# B&R Automation Studio project RS15_RX_30005_r00 (part 4)

#### FP_HeaterInit.st
```iecst
(********************************************************************
 * COPYRIGHT -- .
 ********************************************************************
 * Program: FP_Heater
 * File: FP_HeaterInit.st
 * Author: dominique
 * Created: August 22, 2012
 ********************************************************************
 * Implementation of program FP_Heater
 ********************************************************************)

PROGRAM _INIT

  rPT1_t                   := 25 ;
  rDeltaTStopPicChauf      := 68 ;
  rSeuilConsTempActBattTOR := 132.8 ;

  rPIDRegTChaufKP[1] := 18 ;
  rPIDRegTChaufKI[1] := 30 ;
  rPIDRegTChaufKD[1] := 1 ;

END_PROGRAM
```

### Program Logical/BagMachine_Section/GlobProgCalc (IEC)

#### GlobProgCalcCyclic.st - Cyclic code
```iecst
(********************************************************************
 * COPYRIGHT -- .
 ********************************************************************
 * Program: GlobProgCalc
 * File: GlobProgCalcCyclic.st
 * Author: dominique
 * Created: October 27, 2011
 ********************************************************************
 * Implementation of program GlobProgCalc
 ********************************************************************)

PROGRAM _CYCLIC
// --------------------------------------------------------------------------------------------------
  // Tube Length Limit

  CASE g_iMachType OF
    C_iRS15 :
      g_rMaxBagSize_Inch := g_rMaxBagSize_RS15_mm / 25.4 ;
      g_rMinBagSize_Inch := g_rMinBagSize_RS15_mm / 25.4 ;
    C_iRS26 :
      IF gRecipeActive.bSelEnvBProd THEN
        // Case Envelope Bag
        g_rMaxBagSize_Inch := g_rMaxBagSize_EnvB_mm / 25.4 ;
        g_rMinBagSize_Inch := g_rMinBagSize_EnvB_mm / 25.4 ;
      ELSE
        g_rMaxBagSize_Inch := g_rMaxBagSize_RS26_mm / 25.4 ;
        g_rMinBagSize_Inch := g_rMinBagSize_RS26_mm / 25.4 ;
      END_IF ;
  END_CASE ;

  // Limit operator setting in case of Flexo Type
  gRecipeActive.iPrintUp := LIMIT(1,gRecipeActive.iPrintUp,4) ;
  gRecipeActive.Repeat := LIMIT(g_rMinBagSize_Inch,gRecipeActive.Repeat,g_rMaxBagSize_Inch) ;

  // Repeat calculation in case of Flexo Press
  rPrintUp := INT_TO_REAL(gRecipeActive.iPrintUp) ; // Number of pictures per round of printing cylinder
  CASE g_iFlexoType OF
    C_iM : ; // Case Metric
      iNmaxTooth := TRUNC(g_rMaxBagSize_Inch*25.4/10.0) ;
      iNminTooth := TRUNC(g_rMinBagSize_Inch*25.4/10.0) ;
      IF gRecipeActive.bSelFPProd THEN
        gRecipeActive.Repeat := TRUNC(gRecipeActive.iNumToothGearPrint*10.0)/25.4/rPrintUp ;
      ELSE
        // treatment imperfection calculation of number of tooth otherwise 600mm give 59 tooth instead of 60
        rRepeatMetric := gRecipeActive.Repeat * 25.4 ;
        rRepMet_DecPart := rRepeatMetric - TRUNC(rRepeatMetric) ;
        IF rRepMet_DecPart > 0.5 THEN
          gRecipeActive.iNumToothGearPrint := TRUNC(rRepeatMetric/10.0) + 1 ;
        ELSE
          gRecipeActive.iNumToothGearPrint := TRUNC(rRepeatMetric/10.0) ;
        END_IF ;
      END_IF
      gRecipeActive.iNumToothGearPrint := LIMIT(iNminTooth,gRecipeActive.iNumToothGearPrint,iNmaxTooth) ;
    C_i8DP : ; // Case 8DP
      iNmaxTooth := TRUNC(g_rMaxBagSize_Inch/3.14*8.0) ;
      iNminTooth := TRUNC(g_rMinBagSize_Inch/3.14*8.0) ;
      IF gRecipeActive.bSelFPProd THEN
        gRecipeActive.Repeat := TRUNC(gRecipeActive.iNumToothGearPrint*PI/8.0*1000.0)/1000.0/rPrintUp ;
      ELSE
        gRecipeActive.iNumToothGearPrint := TRUNC(gRecipeActive.Repeat/3.14*8.0) ;
      END_IF
      gRecipeActive.iNumToothGearPrint := LIMIT(iNminTooth,gRecipeActive.iNumToothGearPrint,iNmaxTooth) ;
    C_i10DP : ; // Case 10DP
      iNmaxTooth := TRUNC(g_rMaxBagSize_Inch/3.14*10.0) ;
      iNminTooth := TRUNC(g_rMinBagSize_Inch/3.14*10.0) ;
      IF gRecipeActive.bSelFPProd THEN
        gRecipeActive.Repeat := TRUNC(gRecipeActive.iNumToothGearPrint*PI/10.0*1000.0)/1000.0/rPrintUp ;
      ELSE
        gRecipeActive.iNumToothGearPrint := TRUNC(gRecipeActive.Repeat/3.14*10.0) ;
      END_IF
      gRecipeActive.iNumToothGearPrint := LIMIT(iNminTooth,gRecipeActive.iNumToothGearPrint,iNmaxTooth) ;
    C_i1_4P : ; // Case 1/4"
      iNmaxTooth := TRUNC(g_rMaxBagSize_Inch*4.0) ;
      iNminTooth := TRUNC(g_rMinBagSize_Inch*4.0)+1 ; // D.M. 16/11/2011 RS26 BrownPaper_14606 +1 otherwise minimum tube lentgth = 159mm insted of 160mm and it important for the synchro ratio of the Holding Axis lower than tube length 160mm the Holding Axis makes 1/4 round per bag => not correct for RS26
      IF gRecipeActive.bSelFPProd THEN
        gRecipeActive.Repeat := TRUNC(gRecipeActive.iNumToothGearPrint/4.0*1000.0)/1000.0/rPrintUp ;
      ELSE
        gRecipeActive.iNumToothGearPrint := TRUNC(gRecipeActive.Repeat*4.0) ;
      END_IF
      gRecipeActive.iNumToothGearPrint := LIMIT(iNminTooth,gRecipeActive.iNumToothGearPrint,iNmaxTooth) ;
  END_CASE

// --------------------------------------------------------------------------------------------------
  // Synchro axis OK
  g_bSynchroAxisOK := ( gA[1].Ind_bSynchroOK  AND
                        gA[11].Ind_bSynchroOK OR
                        NOT(gPerf_On) )       AND
                      ( gA[2].Ind_bSynchroOK  OR
                        NOT(gA[2].bActive) )  AND
                      gA[3].Ind_bSynchroOK    AND
                      gA[4].Ind_bSynchroOK    AND
                      gA[5].Ind_bSynchroOK    AND
                      gA[6].Ind_bSynchroOK    AND
                      gA[7].Ind_bSynchroOK    AND
                      ( gA[8].Ind_bSynchroOK  OR
                        NOT(gA[8].bActive) )  AND
                      ( gA[12].Ind_bSynchroOK OR
                        NOT(gA[12].bInMach) ) AND
                      ( gA[13].Ind_bSynchroOK OR
                        NOT(gA[13].bInMach) ) AND
                      1                       ;
  // Synchro axis in progress
  g_bSynchroAxisInProgress := gA[9].Ind_InMotion    AND
                              NOT(g_bSynchroAxisOK) ;
  //
  // Synchro Holding, Tearing and Drum axis
  g_bIndSynchroHTD_OK := gA[3].Ind_bSynchroOK    AND
                         gA[4].Ind_bSynchroOK    AND
                         gA[7].Ind_bSynchroOK    AND
                         ( gA[12].Ind_bSynchroOK OR
                           NOT(gA[12].bInMach) ) AND
                         ( gA[13].Ind_bSynchroOK OR
                           NOT(gA[13].bInMach) ) ;

// --------------------------------------------------------------------------------------------------
  g_bCycManTimeSetOn := gstCycA[1].CycManTimSet.bSCyc  OR
                        gstCycA[3].CycManTimSet.bSCyc  OR
                        gstCycA[4].CycManTimSet.bSCyc  OR
                        gstCycA[7].CycManTimSet.bSCyc  OR
                        gstCycA[12].CycManTimSet.bSCyc AND
                        gA[12].bInMach                 OR
                        gstCycA[13].CycManTimSet.bSCyc AND
                        gA[13].bInMach                 OR
                        0                              ;
END_PROGRAM
```

#### GlobProgCalc.var - Local variables
```iecst
(********************************************************************
 * COPYRIGHT -- .
 ********************************************************************
 * Program: GlobProgCalc
 * File: GlobProgCalc.var
 * Author: dominique
 * Created: October 27, 2011
 ********************************************************************
 * Local variables of program GlobProgCalc
 ********************************************************************)

VAR
  rPrintUp      : REAL ;
  rRepeatMetric : REAL ;
  iNmaxTooth    : INT ;
  iNminTooth    : INT ;
  rRepMet_DecPart : REAL ;
END_VAR

VAR CONSTANT

END_VAR
```

### Program Logical/BagMachine_Section/Holding/Axis3/A3_Automat

#### A3_Automat.var
```iecst
(********************************************************************
 * COPYRIGHT -- Microsoft
 ********************************************************************
 * Program: A3_Automat
 * File: A3_Automat.var
 * Author: pkiel
 * Created: July 13, 2011
 ********************************************************************
 * Local variables of program A3_Automat
 ********************************************************************)
VAR
	AutData : MC_AUTDATA_TYP;
	AutomatStart : BOOL;
	ErrorID : UINT;
	MasterParID : UINT;
	MC_BR_AutControl_0 : MC_BR_AutControl;
  uiMC_BR_AutControl_0_MemoErrorID : UINT := 0 ;
	MC_BR_InitMasterParIDTransfer_0 : MC_BR_InitMasterParIDTransfer;
	ParID_Ready : BOOL;
	PeriodDint : DINT;
	Position_Dint : DINT;
	PositionDint : DINT;
	PositionMOD : DINT;
	PositionOffset : DINT;
	RepeatMetric : INT;
	Slave_AdjustedPosition : REAL;
	Slave_AxisPeriod : REAL;
	SlaveStartOffset : REAL;
	Synch_Request : BOOL;
	ToolCount_2 : BOOL;
  bTest_ : ARRAY[0..9] OF  BOOL;
  iTest_ : ARRAY[0..9] OF  INT;
  rTest_ : ARRAY[0..9] OF  REAL;
  rMaCompDist : REAL ;
  rSPMaPos    : REAL ;
  rOffsetDeg  : REAL ;
  rSlCompDist : REAL ;
  rTemp_      : ARRAY[0..9] OF REAL ;
  usiMemoStat : USINT;
  bEDGEPOS : BOOL ;
  rRepeatMetric : REAL ;
END_VAR
```

#### A3_AutomatCyclic.st
```iecst
(********************************************************************
 * COPYRIGHT -- Microsoft
 ********************************************************************
 * Program: A3_Automat
 * File: A3_AutomatCyclic.st
 * Author: pkiel
 * Created: July 13, 2011
 ********************************************************************
 * Implementation of program A3_Automat
 ********************************************************************)

PROGRAM _CYCLIC

(**** STRAIGHT GEARED CAM AUTOMAT WITH ABSOLUTE PHASE SYNCHRONIZATION FOR HOLDING AXIS ***)

(* Set Up Master Position Parameter ID *)

  // Holding timing setting
  MC_BR_AutControl_0.Signal1 := 0 ;
  MC_BR_AutControl_0.Signal2 := 0 ;

  IF gstCycA[3].CycManTimSet.CmdSynchroOn       AND
     (MC_BR_AutControl_0.ActualStateIndex <> 3) THEN
    MC_BR_AutControl_0.Signal1 := 1 ;
  END_IF

  IF NOT(gstCycA[3].CycManTimSet.CmdSynchroOn) AND
     (MC_BR_AutControl_0.ActualStateIndex = 3) THEN
      MC_BR_AutControl_0.Signal2 := 1 ;
  END_IF

  // A3 Synchro OK indicator
  gstCycA[3].CycManTimSet.bSynchroOkSlavA[3] := ( MC_BR_AutControl_0.ActualStateIndex = 3 )  AND
                                                gA[3].Ind_SynchronizedMotion AND ParID_Ready ;

  //Synch_Request := gA[3].Cmd_SynchronizedMotion ;
  Synch_Request := gA[3].Cmd_SynchronizedMotion AND NOT(MC_BR_AutControl_0.Stop) ;  // D.M. 26/01/2012 RS26 Pyrollpack_14661 added because it happened that Stop=1 and Synch_Request=1 => MC_BR_AutControl_0 makes fault 29256
	IF (Synch_Request AND NOT ParID_Ready) THEN
		MC_BR_InitMasterParIDTransfer_0.Master:=gA[9].Ident;
    MC_BR_InitMasterParIDTransfer_0.Slave:=gA[3].Ident;
    MC_BR_InitMasterParIDTransfer_0.MasterParID:=412;
    MC_BR_InitMasterParIDTransfer_0.SlaveChannel:=0;
    MC_BR_InitMasterParIDTransfer_0.Execute:=TRUE;
    IF (MC_BR_InitMasterParIDTransfer_0.Done) THEN
      MasterParID:=MC_BR_InitMasterParIDTransfer_0.ReceiveParID;
      MC_BR_InitMasterParIDTransfer_0.Execute:=FALSE;
      ParID_Ready:=1;
    ELSIF (MC_BR_InitMasterParIDTransfer_0.Error) THEN
    (*Store ErrorID in a variable,
      ErrorID is reset on falling edge of 'Execute'*)
      ErrorID:=MC_BR_InitMasterParIDTransfer_0.ErrorID;
      ParID_Ready:=0;
      MC_BR_InitMasterParIDTransfer_0.Execute:=FALSE;
	    END_IF
	END_IF
	MC_BR_InitMasterParIDTransfer_0();

(**** Initialize Automat Parameters Upon Automat Start Request ****)
	IF (EDGEPOS(ParID_Ready))THEN

		(* Slave Axis Period Based On Number Of Tools On Maintaining Shaft *)
		(* Number of Tools On Holding (Maintaining) Shaft Based On Tube Length...Lengh>160m = 2 Tools, Length<=160mm = 4 Tools *)
			rRepeatMetric := gRecipeActive.Repeat*25.4;
      Slave_AxisPeriod := gA[3].AxisPeriod * gA[3].rRSynNum/gA[3].rRSynDen;
      PeriodDint := REAL_TO_DINT(Slave_AxisPeriod);
      PositionDint := REAL_TO_DINT(gA[3].PositionCount);
      Slave_AdjustedPosition := (DINT_TO_REAL(PeriodDint-(PositionDint MOD PeriodDint)))*gA[3].UnitsPerInch;

		(**** Calculate Slave Start Offset ****)
			PositionOffset:= REAL_TO_DINT((gA[9].PositionInch-(gA[3].PositionInch-gRecipeActive.Holding_Offset))*1000);
			PositionMOD:= REAL_TO_DINT(gRecipeActive.Repeat*1000);
			SlaveStartOffset:= (DINT_TO_REAL(PositionOffset MOD PositionMOD))/1000;
			IF (SlaveStartOffset >= (0.5*gRecipeActive.Repeat)) THEN
				SlaveStartOffset := SlaveStartOffset - gRecipeActive.Repeat;
			END_IF
			IF (SlaveStartOffset < (-0.5*gRecipeActive.Repeat)) THEN
				SlaveStartOffset := SlaveStartOffset + gRecipeActive.Repeat;
			END_IF

      rTemp_[1] := gA[3].PositionDeg ;
      rTemp_[2] := gA[9].PositionDeg ;

      rOffsetDeg := gRecipeActive.rHolding_PhasMasterDeg ;

      rSPMaPos := (gA[3].PositionDeg - rOffsetDeg)/(gA[3].rRSynNum/gA[3].rRSynDen) ;
      rTemp_[0] := rSPMaPos - gA[9].PositionDeg ;

      rMaCompDist := H_FC_Modulus (
                          //IN_rMod := (360 * gA[3].rRSynNum/gA[3].rRSynDen) ,
                          IN_rMod := 360 ,
                          IN_rVar := rTemp_[0]
                                  ) ;

		(*general automat parameter*)
			//AutData.Master				  := gA[3].Ident;
			AutData.MasterParID			  := MasterParID;
			AutData.StartPosition		  := 0;
			AutData.StartInterval		  := gA[9].AxisPeriod;
			AutData.MaxMasterVelocity	:= gr_rMachMaxSpeed_BPM ;

		(*Automat STATE 0 Basis State*)
			AutData.State[0].Event[0].Type		  := ncST_END;
			AutData.State[0].Event[0].Attribute	:= ncAT_ONCE;
      IF (rMaCompDist >= 1/gA[3].UnitsPerDeg) AND
         gA[3].bSynchroReq                    THEN
        AutData.State[0].Event[0].NextState := 1;
      ELSE
        rMaCompDist := 1/gA[3].UnitsPerDeg ;
        AutData.State[0].Event[0].NextState := 2;
      END_IF

    //Automat STATE 0 Basis State
      AutData.State[0].Event[0].Type      := ncST_END;
      AutData.State[0].Event[0].Attribute := ncAT_ONCE;
      AutData.State[0].Event[0].NextState := 1;

    //Automat STATE 1 Master/Slave Absolute Phase Correction
      AutData.State[1].CamProfileIndex := 16#FFFF;
      AutData.State[1].MasterFactor    := REAL_TO_UDINT(rMaCompDist * gA[3].UnitsPerDeg) ;
      AutData.State[1].SlaveFactor     := 0 ;
      AutData.State[1].CompMode        := ncOFF;

      AutData.State[1].Event[0].Type      := ncST_END;
      AutData.State[1].Event[0].Attribute := ncST_END;
      AutData.State[1].Event[0].NextState := 2;

      AutData.State[1].Event[1].Type      := ncSIGNAL1 ;
      AutData.State[1].Event[1].Attribute := ncAT_ONCE ;
      AutData.State[1].Event[1].NextState := 3 ;

    //Automat STATE 2 Master/Slave run
      AutData.State[2].CamProfileIndex := 16#FFFF;
      AutData.State[2].MasterFactor    := REAL_TO_UDINT(gA[9].AxisPeriod) ;
      AutData.State[2].SlaveFactor     := REAL_TO_UDINT(Slave_AxisPeriod) ;
      AutData.State[2].CompMode        := ncOFF;

      AutData.State[2].Event[0].Type      := ncST_END ;
      AutData.State[2].Event[0].Attribute := ncST_END ;
      AutData.State[2].Event[0].NextState := 2 ;

      AutData.State[2].Event[1].Type      := ncST_END+ncNEGATIVE ;
      AutData.State[2].Event[1].Attribute := ncST_END ;
      AutData.State[2].Event[1].NextState := 2 ;

      AutData.State[2].Event[2].Type      := ncSIGNAL1 ;
      AutData.State[2].Event[2].Attribute := ncAT_ONCE ;
      AutData.State[2].Event[2].NextState := 3 ;

    //Automat STATE 3 Master/Slave Timing setting
      AutData.State[3].CamProfileIndex := 16#FFFF;
      AutData.State[3].MasterFactor    := REAL_TO_UDINT(gA[9].AxisPeriod) ;
      AutData.State[3].SlaveFactor     := REAL_TO_UDINT(Slave_AxisPeriod) ;
      AutData.State[3].CompMode        := ncOFF;

      AutData.State[3].Event[0].Type      := ncST_END ;
      AutData.State[3].Event[0].Attribute := ncST_END ;
      AutData.State[3].Event[0].NextState := 3 ;

      AutData.State[3].Event[1].Type      := ncST_END+ncNEGATIVE ;
      AutData.State[3].Event[1].Attribute := ncST_END ;
      AutData.State[3].Event[1].NextState := 3 ;

      AutData.State[3].Event[2].Type      := ncSIGNAL2 ;
      AutData.State[3].Event[2].Attribute := ncAT_ONCE ;
      AutData.State[3].Event[2].NextState := 2 ;

			MC_BR_AutControl_0.Enable 		  := 1;
			MC_BR_AutControl_0.AdrAutData 	:= ADR(AutData);
			MC_BR_AutControl_0.InitAutData 	:= 1;
	END_IF
			(* wait for initialization done or restart *)
			IF ((MC_BR_AutControl_0.AutDataInitialized=1) AND (Synch_Request)) THEN
				MC_BR_AutControl_0.InitAutData := 0;
				MC_BR_AutControl_0.Enable :=1 ;
        uiMC_BR_AutControl_0_MemoErrorID := 0 ;
				AutomatStart := 1;;
			END_IF
			(* check if error occured *)
			IF (MC_BR_AutControl_0.ErrorID <> 0) THEN
				MC_BR_AutControl_0.Enable := 0;
        uiMC_BR_AutControl_0_MemoErrorID := MC_BR_AutControl_0.ErrorID ;
			END_IF

	(******************** ENABLE CAM-AUTOMAT **********************)

	IF (AutomatStart) THEN
			MC_BR_AutControl_0.Start := 1;
			AutomatStart := 0;
	END_IF

	IF (NOT Synch_Request) THEN
			MC_BR_AutControl_0.Stop := 1;
			MC_BR_AutControl_0.Start := 0;
			ParID_Ready := 0;
			IF (MC_BR_AutControl_0.Running=0) THEN
				MC_BR_AutControl_0.Enable := 0;
				MC_BR_AutControl_0.Stop := 0;
			END_IF
   //*************************************************
   // D.M. 26/01/2012 RS26 Pyrollpack_14661 added because after guard fault it happened that Stop=1 and MC_BR_AutControl_0.Enable => not possible to finish MC_BR_AutControl_0 => program locked
      IF MC_BR_AutControl_0.Stop        AND
         NOT(MC_BR_AutControl_0.Enable) THEN
        MC_BR_AutControl_0.Enable := 1 ;
      END_IF
   //*************************************************
	END_IF

	gA[3].Ind_AutomatEnabled:=MC_BR_AutControl_0.Enable;
	gA[3].Ind_CurrentAutomatState:=MC_BR_AutControl_0.ActualStateIndex;
  gA[3].Ind_bSynchroOK := (MC_BR_AutControl_0.ActualStateIndex >= 2) AND gA[3].Ind_SynchronizedMotion ;

	(********************** MC_AUTCONTROL *************************)
	MC_BR_AutControl_0.Slave:= gA[3].Ident;
	MC_BR_AutControl_0();

END_PROGRAM
```

### Program Logical/BagMachine_Section/Holding/Axis3/A3_Basic

#### A3_BasicCyclic.st
```iecst
(********************************************************************
 * COPYRIGHT -- Microsoft
 ********************************************************************
 * Program: A3_Basic
 * File: A3_BasicCyclic.st
 * Author: pkiel
 * Created: July 13, 2011
 ********************************************************************
 * Implementation of program A3_Basic
 ********************************************************************)

PROGRAM _CYCLIC

	gA[3].UnitsPerInch := gA[3].AxisPeriod/gRecipeActive.Repeat;
  gA[3].InchPerDeg := gA[3].UnitsPerDeg / gA[3].UnitsPerInch ;
  gA[3].rRSynNum := 1 ;
  rRepeatMetric := gRecipeActive.Repeat*25.4;
  IF (rRepeatMetric>=gr_rBagSize2_4Hold_mm) THEN
    IF (g_rNumbPliers <> 0) THEN
      gA[3].rRSynDen := g_rNumbPliers / 2.0 ;
    ELSE
      gA[3].rRSynDen := 2.0 ;
    END_IF
  ELSE
    gA[3].rRSynDen := 4.0 ;
  END_IF

  // Case Envelope Bag
  IF gRecipeActive.bSelEnvBProd THEN
    IF (rRepeatMetric<=gr_rBagSize1_2Hold_mm) THEN
      gA[3].rRSynDen := 2.0 ;
    ELSE
      gA[3].rRSynDen := 1.0 ;
    END_IF
  END_IF

  // Axis inside contact zone
  IF (gA[3].rRSynDen <> 0.0) THEN
    rA3PosTempAxis_deg := H_FC_Modulus (
                                IN_rMod := (360 * gA[3].rRSynNum/gA[3].rRSynDen) ,
                                IN_rVar := gA[3].PositionDeg
                                        ) ;
  END_IF
  gA[3].Ind_bInContactZone := (rA3PosTempAxis_deg <= gr_rHoldAxContactZone) ;

	IF (gA[3].Ident<>0) THEN

	(************************ READ DRIVE STATUS *************************)
	(* Access to the following bools:
	gA[x]_DriveStatus.Simulation			: If TRUE, simulation mode is active
	gA[x]_DriveStatus.NetworkInit			: If TRUE, the network is initialized
	gA[x]_DriveStatus.HomeSwitch			: If TRUE, the digital reference switch input is active
	gA[x]_DriveStatus.PosHWSwitch			: If TRUE, the positive hardware end switch is active
	gA[x]_DriveStatus.NegHWSwitch			: If TRUE, the negative hardware end switch is active
	gA[x]_DriveStatus.Trigger1				: If TRUE, the first trigger input is active
	gA[x]_DriveStatus.Trigger2				: If TRUE, the second trigger input is active
	gA[x]_DriveStatus.DriveEnable			: If TRUE, the enable input is active
	gA[x]_DriveStatus.ControllerReady		: If TRUE, the controller is ready to beturned on
	gA[x]_DriveStatus.ControllerStatus		: If TRUE, the controller is turned on (Same as MC_Power.Status)
	gA[x]_DriveStatus.AxisError				: If TRUE, at least one error has occurred (not acknowledged)
	gA[x]_DriveStatus.LagWarning			: If TRUE, the lag error has exceeded the limit value specified for a warning*)
		MC_BR_ReadDriveStatus_0.Enable := 1;
		MC_BR_ReadDriveStatus_0.Axis := gA[3].Ident;
		MC_BR_ReadDriveStatus_0.AdrDriveStatus := ADR (DriveStatus);
		MC_BR_ReadDriveStatus_0();
		gA[3].Ind_Simulation		:=	DriveStatus.Simulation;
		gA[3].Ind_NetworkInit		:=	DriveStatus.NetworkInit;
		gA[3].Input_Home			:=	DriveStatus.HomeSwitch;
		gA[3].Input_PosHW			:=	DriveStatus.PosHWSwitch;
		gA[3].Input_NegHW			:=	DriveStatus.NegHWSwitch;
		gA[3].Input_Trigger1		:=	DriveStatus.Trigger1;
		gA[3].Input_Trigger2		:=	DriveStatus.Trigger2;
		gA[3].Input_DriveEnable		:=	DriveStatus.DriveEnable;
		gA[3].Ind_ControllerReady	:=	DriveStatus.ControllerReady;
		gA[3].Ind_ControllerStatus	:=	DriveStatus.ControllerStatus;
		gA[3].Error					:=	DriveStatus.AxisError;
		gA[3].Ind_LagWarning		:=	DriveStatus.LagWarning;

	(************************ READ AXIS ERROR **********************)
		MC_ReadAxisError_0.Enable := gA[3].Ind_NetworkInit;
		MC_ReadAxisError_0.Axis := gA[3].Ident;
		MC_ReadAxisError_0.DataAddress := ADR(gA[3].ErrorText);
		MC_ReadAxisError_0.DataLength := SIZEOF(gA[3].ErrorText);
		MC_ReadAxisError_0.DataObjectName := 'Error_Eng';
		MC_ReadAxisError_0();
		IF(MC_ReadAxisError_0.Valid) THEN
			gA[3].ErrorID := MC_ReadAxisError_0.AxisErrorID;
			gA[3].ErrorCount := MC_ReadAxisError_0.AxisErrorCount;
		END_IF
	(* Auto Acknowledge Errors *)
		IF (gA[3].Cmd_Reset AND (gA[3].ErrorCount<>0) AND NOT AutoAck) THEN
			AutoAck:=1;
		ELSE
			AutoAck:=0;
		END_IF
	(*Axis Error Acknowledge*)
		IF (EDGEPOS(AutoAck) OR EDGEPOS(gA[3].ErrorAck)) THEN
			MC_ReadAxisError_0.Acknowledge := 1;
		ELSE;
			MC_ReadAxisError_0.Acknowledge :=0;
		END_IF

	(************************ RESET AXIS ERROR **********************)
		IF (gA[3].Cmd_Reset AND (gA[3].ErrorCount=0) AND gA[3].ErrorStop) THEN
			MC_Reset_0.Execute:=1;
		END_IF
		IF (MC_Reset_0.Done) THEN
			MC_Reset_0.Execute:=0;
			gA[3].Cmd_Reset:=0;
			ResetError := 0;
		END_IF
		IF (MC_Reset_0.Error) THEN
			MC_Reset_0.Execute:=0;
			gA[3].Cmd_Reset:=0;
			ResetError := 1;
		END_IF
		MC_Reset_0.Axis:=gA[3].Ident;
		MC_Reset_0();

	(************************ READ AXIS STATUS *************************)
		MC_ReadStatus_0.Enable := gA[3].Ind_NetworkInit;
		MC_ReadStatus_0.Axis := gA[3].Ident;
		MC_ReadStatus_0();
		IF(MC_ReadStatus_0.Valid = TRUE)THEN
			gA[3].Ind_Enabled 			:= NOT (MC_ReadStatus_0.Disabled);
			gA[3].Ind_StandStill		:= MC_ReadStatus_0.StandStill;
			gA[3].Ind_Stopping			:= MC_ReadStatus_0.Stopping;
			gA[3].Ind_DiscreteMotion	:= MC_ReadStatus_0.DiscreteMotion;
			gA[3].Ind_ContinuousMotion	:= MC_ReadStatus_0.ContinuousMotion;
			gA[3].Ind_SynchronizedMotion:= MC_ReadStatus_0.SynchronizedMotion;
			gA[3].ErrorStop				:= MC_ReadStatus_0.Errorstop;
		END_IF
    IF NOT(gA[3].Ind_Enabled) THEN
      gA[3].bSynchroReq := 1 ;
    END_IF
    IF EDGEPOS(gA[3].Ind_bSynchroOK) THEN
      gA[3].bSynchroReq := 0 ;
    END_IF

	(******************** INIT POSITION MODULUS  *********************)
		MC_BR_InitModPos_0.Execute:= InitModPosition;
		MC_BR_InitModPos_0.Axis:= gA[3].Ident;
		MC_BR_InitModPos_0.Period:= REAL_TO_UDINT(gA[3].AxisPeriod);
		MC_BR_InitModPos_0.Factor:=1;
		InitModPos_Done:=MC_BR_InitModPos_0.Done;
		MC_BR_InitModPos_0();

	(******************** INIT ENDLESS POSITION *********************)
		MC_BR_InitEndlessPosition_0.Execute:= InitModPos_Done;
		MC_BR_InitEndlessPosition_0.Axis:= gA[3].Ident;
		MC_BR_InitEndlessPosition_0.DataAddress:= ADR(gEndPosData[3]);
		IF (MC_BR_InitEndlessPosition_0.Done) THEN
			InitModPosition:=0;
			InitEndlessPosition:=0;
			HomeRestore:=1;
		END_IF
		MC_BR_InitEndlessPosition_0();

	(************************ HOME AXIS FIRST POWER UP **********************)
		IF (HomeRestore AND NOT gA3_FirstHomed) THEN
			MC_Home_0.Execute:=1;
		END_IF
		MC_Home_0.Axis:=gA[3].Ident;
		MC_Home_0.Position:=0;
		MC_Home_0.HomingMode:=mcHOME_DIRECT;
		IF (MC_Home_0.Done) THEN
			MC_Home_0.Execute:=0;
			gA3_FirstHomed:=1;
		END_IF
		MC_Home_0();

	(************************ HOME AXIS **********************)
		IF (gA3_FirstHomed) THEN
			MC_Home_1.Execute:=HomeRestore;
		END_IF
		MC_Home_1.Axis:=gA[3].Ident;
		MC_Home_1.Position:=0;
		MC_Home_1.HomingMode:=mcHOME_RESTORE_POS;
		IF (MC_Home_1.Done) THEN
			gA[3].Ind_Homed:=1;
			HomeRestore:=0;
		END_IF
		MC_Home_1();

	(******************** READ ACTUAL POSITION *********************)
		MC_ReadActualPosition_0.Enable:= gA[3].Ind_NetworkInit;
		MC_ReadActualPosition_0.Axis:= gA[3].Ident;
		MC_ReadActualPosition_0();
		IF(MC_ReadActualPosition_0.Valid = TRUE)THEN
			gA[3].PositionCount := MC_ReadActualPosition_0.Position;
			gA[3].PositionInch := gA[3].PositionCount/gA[3].UnitsPerInch;
			gA[3].PositionDeg := gA[3].PositionCount/gA[3].UnitsPerDeg;
    END_IF

  (******************** HOLDING IN CONTACT ZONE *********************)
    rTempPosHolding  := H_FC_Modulus (
                             IN_rMod := 360 * gA[3].rRSynNum / gA[3].rRSynDen ,
                             IN_rVar := gA[3].PositionDeg
                                     ) ;
    gA[3].Ind_bInContactZone := (rTempPosHolding < gr_rHoldAxContactZone) ;

  //******************** READ SET POINT POSITION *********************
    // Slave side  : ParID 428 SGEN_S_SET : CTRL Position controller: Input set position
    // Master side : ParID 412 S_SET_VAX1 : 412: VAX: Position

    // Slave side
    MC_BR_CyclicRead_0.Axis        := gA[3].Ident ;
    MC_BR_CyclicRead_0.Enable      := gA[3].Ind_NetworkInit;
    MC_BR_CyclicRead_0.ParID       := 428 ;
    MC_BR_CyclicRead_0.DataAddress := ADR(iiSP_SlPos_U);
    MC_BR_CyclicRead_0.DataType    := ncPAR_TYP_DINT ;
    // Master side
    MC_BR_CyclicRead_1.Axis        := gA[9].Ident ;
    MC_BR_CyclicRead_1.Enable      := gA[3].Ind_NetworkInit;
    MC_BR_CyclicRead_1.ParID       := 412 ;
    MC_BR_CyclicRead_1.DataAddress := ADR(iiSP_MaPos_U);
    MC_BR_CyclicRead_1.DataType    := ncPAR_TYP_DINT ;

    IF MC_BR_CyclicRead_0.Valid THEN
      rSP_SlPos_Deg := iiSP_SlPos_U/gA[3].UnitsPerDeg ;
    ELSIF MC_BR_CyclicRead_0.Error THEN
      MC_BR_CyclicRead_0.Enable := 0 ;
    END_IF
    IF MC_BR_CyclicRead_1.Valid THEN
      rSP_MaPos_Deg := iiSP_MaPos_U/gA[9].UnitsPerDeg ;
    ELSIF MC_BR_CyclicRead_1.Error THEN
      MC_BR_CyclicRead_1.Enable := 0 ;
    END_IF
    MC_BR_CyclicRead_0();
    MC_BR_CyclicRead_1();

  //******************** READ ACTUAL OFFSET *********************
  IF gA[3].rRSynDen > 0.0 THEN
    rTempActPhasDeg := rSP_SlPos_Deg - gA[3].rRSynNum / gA[3].rRSynDen * rSP_MaPos_Deg ;
    gA[3].rActPhasDeg := H_FC_Modulus (
                             IN_rMod := 360 * gA[3].rRSynNum / gA[3].rRSynDen ,
                             IN_rVar := rTempActPhasDeg
                                      ) ;
  END_IF

	(******************** READ ACTUAL VELOCITY *********************)
		IF(MC_ReadActualVelocity_0.Error=TRUE) THEN
			MC_ReadActualVelocity_0.Enable:= 0;
		ELSE
			MC_ReadActualVelocity_0.Enable:= 1;
		END_IF
		MC_ReadActualVelocity_0.Axis:= gA[3].Ident;
		MC_ReadActualVelocity_0();
		IF(MC_ReadActualVelocity_0.Valid = TRUE)THEN
//			gA[3].ActualVelocity := MC_ReadActualVelocity_0.Velocity*60/gA[3].SP_MotorPPR;
      gA[3].ActualVelocity := MC_ReadActualVelocity_0.Velocity*60/gA[3].AxisPeriod ; // D.M. 03/08/2011 BrownPaper_14542  Need speed of the axis and not of the shaft of the motor
			IF ABS(gA[3].ActualVelocity>1) THEN // D.M. 03/08/2011 BrownPaper_14542 Add ABS because in case negative velocity Ind_InMotion = 0 instead of 1
				gA[3].Ind_InMotion:=1;
			ELSE
				gA[3].Ind_InMotion:=0;
			END_IF
		END_IF

	(******************** READ ACTUAL TORQUE *********************)
		IF(MC_ReadActualTorque_0.Error=TRUE) THEN
			MC_ReadActualTorque_0.Enable:= 0;
		ELSE
			MC_ReadActualTorque_0.Enable:= 1;
		END_IF
		MC_ReadActualTorque_0.Axis:= gA[3].Ident;
		MC_ReadActualTorque_0();
		IF(MC_ReadActualTorque_0.Valid = TRUE)THEN
			gA[3].ActualTorque := MC_ReadActualTorque_0.Torque;
		END_IF

	(************************ ENABLE AXIS **********************)
		MC_Power_0.Axis:=gA[3].Ident;
		IF (MC_Power_0.Error=0) THEN
			MC_Power_0.Enable:=gA[3].Cmd_Enable;
		ELSE;
			MC_Power_0.Enable:=0;
		END_IF;
		MC_Power_0();

	(************************ AXIS VELOCITY MOVE **********************)
		MC_MoveVelocity_0.Axis:=gA[3].Ident;
		MC_MoveVelocity_0.Velocity:=gA[3].SP_Velocity*gA[3].AxisPeriod/60;
		MC_MoveVelocity_0.Acceleration:=
		MC_MoveVelocity_0.Deceleration:=gA[3].SP_Decel;
		MC_MoveVelocity_0.Direction:=mcPOSITIVE_DIR;
		IF ((EDGEPOS(gA[3].Cmd_ContinuousMotion)) OR (EDGEPOS(gA[3].Cmd_ContinuousMotionUpdate))) THEN
			MC_MoveVelocity_0.Execute:=1;
		ELSE
			MC_MoveVelocity_0.Execute:=0;
		END_IF
		MC_MoveVelocity_0();

  //************************ AXIS OVERRIDE **********************
    MC_SetOverride_0.Axis      := gA[3].Ident ;
    MC_SetOverride_0.Enable    := gA[3].Cmd_Override ;
    MC_SetOverride_0.VelFactor := gA[3].rSP_OverrideV ;
    MC_SetOverride_0.AccFactor := gA[3].rSP_OverrideA ;
    IF (MC_SetOverride_0.Enabled) OR
       (MC_SetOverride_0.Error)   THEN
      gA[3].Cmd_Override := 0 ;
    END_IF
    MC_SetOverride_0();

	(************************ AXIS STOP **********************)
		MC_Stop_0.Axis:=gA[3].Ident;
		IF (gA[3].Ind_ContinuousMotion AND (NOT gA[3].Cmd_ContinuousMotion) AND gAlarmsOK) THEN
			MC_Stop_0.Deceleration:=gA[3].SP_Decel;
			MC_Stop_0.Execute:=1;
		END_IF
		IF (MC_Stop_0.Done OR MC_Stop_0.CommandAborted OR MC_Stop_0.Error) THEN
			MC_Stop_0.Execute:=0;
		END_IF
		MC_Stop_0();

  (************************  ESTOP **********************)
    MC_Stop_1.Axis:=gA[3].Ident;
    IF EDGEPOS(g_bIndEStopStandstill) THEN
      MC_Stop_1.Deceleration:=gA[3].SP_EStopDecel;
      MC_Stop_1.Execute:=1;
    END_IF;
    IF (MC_Stop_1.Done OR MC_Stop_1.CommandAborted OR MC_Stop_1.Error) THEN
      MC_Stop_1.Execute:=0;
      gA[3].Cmd_EStopDisable := 1 ;
    END_IF;
    IF NOT(g_bIndEStopStandstill) THEN
      gA[3].Cmd_EStopDisable := 0 ;
    END_IF;
    MC_Stop_1();

    //************************ AXIS PHASE CONTROL (Inches) First Step **********************
    IF EDGEPOS(gA[3].Cmd_PhaseOffset) THEN
      rSP_PhaseOffset := gA[3].SP_PhaseOffset ;
    END_IF;

    (************************ SHIFTING PERF CONTROL **********************)
    IF gstCycA[3].CycManTimSet.CmdMov THEN
      g_iArrayBagPerfTear := g_iArrayBagPerfTearNul ;
      g_iCountPerfShift[1] := 0 ;
      g_iCountPerfShift[2] := 0 ;
    END_IF;
    IF NOT(g_bIndSynchroHTD_OK)       OR
       gstCycA[3].CycManTimSet.CmdMov THEN
      g_bCmdShiftA[3]  := 0 ;
      g_bCmdShiftA[4]  := 0 ;
      g_bCmdShiftA[7]  := 0 ;
      g_bCmdShiftA[12] := 0 ;
      g_bCmdShiftA[13] := 0 ;
    END_IF;

    IF (g_iCountPerfShift[1] > 0)                    AND
       (g_iArrayBagPerfTear[g_iNumBagPerfTear] <> 0) THEN
      g_bCmdShiftA[3] := 1 ;
    END_IF
    IF g_bCmdShiftA[3] AND
       g_bMachineRun   THEN
      g_iPerfShiftPos := g_iArrayBagPerfTear[g_iNumBagPerfTear] ;
      //rSP_ShiftHolding := g_iPerfShiftPos * gr_rIncrShiftPerf_mm/25.4 * gA[3].rRSynNum/gA[3].rRSynDen ; // D.M. RS26_Pyrollpack_14661 CAUTION !!! Phasing acts on the master side and not slave side, replaced by the code below
      rSP_ShiftHolding := g_iPerfShiftPos * gr_rIncrShiftPerf_mm/25.4 ;
      g_iArrayBagPerfTear[g_iNumBagPerfTear] := 0 ;
      iTest_[0] := iTest_[0] + 1 ;

      g_iCountPerfShift[1] := g_iCountPerfShift[1] - 1 ;
      g_bCmdShiftA[3] := 0 ;
      g_bCmdShiftA[4] := 1 ;
      g_bCmdShiftA[7] := 1 ;
      g_bCmdShiftA[12] := gA[12].bInMach ;
      g_bCmdShiftA[13] := gA[13].bInMach ;
      gA[3].Cmd_PhaseOffset := 1 ;
    END_IF;

    //************************ AXIS PHASE CONTROL (Inches) Next Step **********************
    MC_BR_Phasing_0.Slave:=gA[3].Ident;
    IF gA[3].Ind_SynchronizedMotion AND NOT(gstCycA[3].CycManTimSet.bSCyc) AND st_TON_0.Q THEN
      MC_BR_Phasing_0.Enable:=1;
    ELSE;
      MC_BR_Phasing_0.Enable:=0;
    END_IF;
    IF (gA[3].Cmd_PhaseOffset)              AND
       ( EDGENEG(gA[3].Ind_bInContactZone)  OR
         gRecipeActive.bSelEnvBProd )       AND
       ( EDGENEG(gA[12].Ind_bInContactZone) OR
         NOT(gRecipeActive.bSelEnvBProd) )  AND
       NOT(gstCycA[3].CycManTimSet.bSCyc)   THEN
      MC_BR_Phasing_0.InitData:=1;
      gA[3].Cmd_PhaseOffset := 0 ;
      rSP_PhaseOffsetVal := rSP_PhaseOffset + rSP_ShiftHolding ;
      // Calculation new phase Holdind/Master
      rTemp_[0] := (rSP_PhaseOffsetVal)/gA[3].InchPerDeg ;
      rTemp_[1] := gRecipeActive.rHolding_PhasMasterDeg + rTemp_[0]*gA[3].rRSynNum/gA[3].rRSynDen ;
      gRecipeActive.rHolding_PhasMasterDeg := H_FC_Modulus (IN_rMod := 360*gA[3].rRSynNum/gA[3].rRSynDen, IN_rVar := rTemp_[1]) ;
      rSP_ShiftHolding := 0.0 ;
      rSP_PhaseOffset := 0.0 ;
    ELSE
      MC_BR_Phasing_0.InitData:=0;
    END_IF
    MC_BR_Phasing_0.Shift               := rSP_PhaseOffsetVal*gA[9].UnitsPerInch;
    MC_BR_Phasing_0.Velocity            := 24*gA[3].AxisPeriod/60;
    MC_BR_Phasing_0.Acceleration        := 2*gA[3].SP_Decel;
    MC_BR_Phasing_0.ApplicationDistance := 0.4*gA[9].AxisPeriod * gA[3].rRSynNum/gA[3].rRSynDen;
    MC_BR_Phasing_0.ApplicationMode     := mcMASTER_DISTANCE_BASED;
    MC_BR_Phasing_0.ShiftMode           := mcRELATIVE;
    MC_BR_Phasing_0();

    (************************ AXIS PHASE CONTROL (Inches) TIMING SETTING **********************)
    IF gstCycA[3].CycManTimSet.bSCyc THEN
      IF gA[3].Cmd_ManuTimSetPlus THEN
        rAxisTimSet_SP_Vel := gr_rAxisTimSet_SP_Vel*gA[9].AxisPeriod/60 / (gA[3].rRSynNum/gA[3].rRSynDen) ;
      ELSE
        rAxisTimSet_SP_Vel := - gr_rAxisTimSet_SP_Vel*gA[9].AxisPeriod/60 / (gA[3].rRSynNum/gA[3].rRSynDen) ;
      END_IF
        rAxisTimSet_SP_Acc := gr_rAxisTimSet_SP_Acc*gA[9].AxisPeriod/60/60 ;
    END_IF

    MC_BR_Phasing_1.Slave                  := gA[3].Ident;
    MC_BR_Phasing_1.Enable                 := gstCycA[3].CycManTimSet.bCyc ;
    MC_BR_Phasing_1.InitData               := gstCycA[3].CycManTimSet.bSCyc ;
    MC_BR_Phasing_1.PerformVelocityControl := gstCycA[3].CycManTimSet.CmdMov ;
    MC_BR_Phasing_1.Velocity               := rAxisTimSet_SP_Vel ;
    MC_BR_Phasing_1.Acceleration           := rAxisTimSet_SP_Acc ;
    MC_BR_Phasing_1.ApplicationMode        := mcVELOCITY_CONTROL ;
    MC_BR_Phasing_1();
    st_TON_0(IN:=NOT(MC_BR_Phasing_1.Enable),PT:=T#200ms) ;

    IF NOT(gstCycA[3].CycManTimSet.CmdMov) AND
       MC_BR_Phasing_1.ShiftAttained       OR
       NOT(gstCycA[3].CycManTimSet.bCyc)   OR
       MC_BR_Phasing_1.Error               AND
       1                                   THEN
      gstCycA[3].CycManTimSet.CmdStop := 0 ;
    END_IF
  END_IF

END_PROGRAM
```

#### A3_BasicInit.st
```iecst
(********************************************************************
 * COPYRIGHT -- Microsoft
 ********************************************************************
 * Program: A3_Basic
 * File: A3_BasicInit.st
 * Author: pkiel
 * Created: July 13, 2011
 ********************************************************************
 * Implementation of program A3_Basic
 ********************************************************************)

PROGRAM _INIT

	(* Axis Setpoint Variables *)
		gA[3].SP_MotorPPR := 24000;
		gA[3].SP_GearBoxInput:= 3;
		gA[3].SP_GearBoxOutput:= 2;
		gA[3].AxisPeriod := (gA[3].SP_MotorPPR*gA[3].SP_GearBoxInput/gA[3].SP_GearBoxOutput);
		gA[3].UnitsPerDeg := gA[3].AxisPeriod/360;
		gA[3].SP_Accel := 0.2*gA[3].AxisPeriod;
		gA[3].SP_Decel := 0.4*gA[3].AxisPeriod;
		gA[3].SP_EStopDecel := 1000.0*gA[3].AxisPeriod; // Stop axis from 1000 tr/min in 1s
		gA[3].HomeVelocity := 6*gA[3].AxisPeriod/60;
    gA[3].rSP_CorPosVel := 0.0 ;
    gA[3].rSP_OverrideV := 1.0 ;
    gA[3].rSP_OverrideA := 1.0 ;
    gA[3].Cmd_EStopDisable := 0 ;

	(* access master axis *)
		AxisErrorNcAccess := ncaccess(ncACP10MAN, ADR('Axis3'), ADR(gA[3].Ident));

	(* Trigger Initialization Of ModPosition *)
		InitModPosition:=1;

  // General parameter init
  gr_rHoldAxContactZone := 22.0 ;
END_PROGRAM
```

### Program Logical/BagMachine_Section/Holding/Axis3/A3_Control (IEC)

#### A3_ControlCyclic.ld - Cyclic code
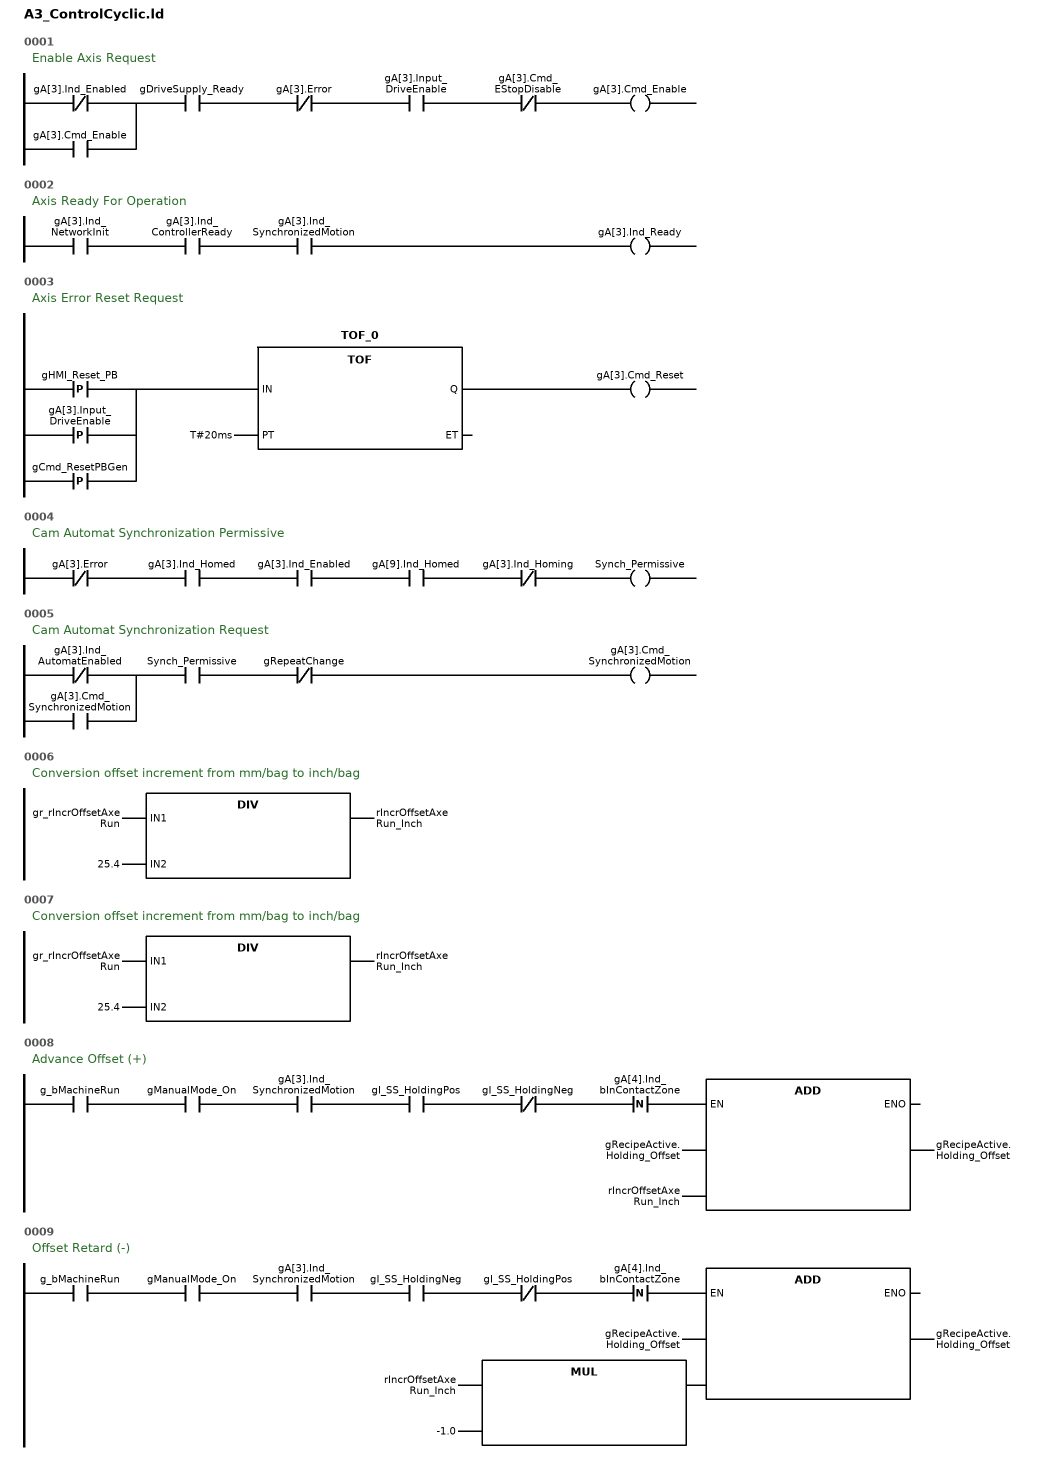
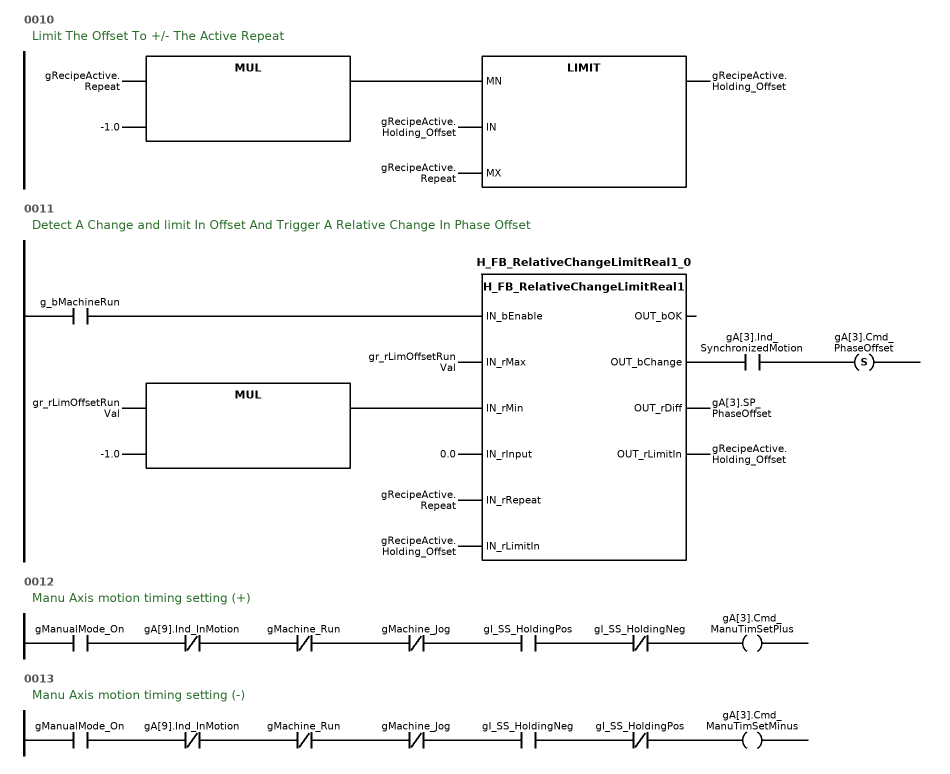
Ladder, written as Structured Text:
```iecst
(********************************************************************
 * COPYRIGHT -- Microsoft
 ********************************************************************
 * Program: A3_Control
 * File: A3_ControlCyclic.ld
 * Author: pkiel
 * Created: July 13, 2011
 ********************************************************************
 * Implementation of program A3_Control
 ********************************************************************)

PROGRAM _CYCLIC
VAR
    _e1 : R_TRIG;
    _e2 : R_TRIG;
    _e3 : R_TRIG;
    _e4 : F_TRIG;
    _e5 : F_TRIG;
END_VAR
(* Network 1: Enable Axis Request *)
gA[3].Cmd_Enable := (NOT gA[3].Ind_Enabled OR gA[3].Cmd_Enable) AND gDriveSupply_Ready AND NOT gA[3].Error AND gA[3].Input_DriveEnable AND NOT gA[3].Cmd_EStopDisable;

(* Network 2: Axis Ready For Operation *)
gA[3].Ind_Ready := gA[3].Ind_NetworkInit AND gA[3].Ind_ControllerReady AND gA[3].Ind_SynchronizedMotion;

(* Network 3: Axis Error Reset Request *)
_e1(CLK := gHMI_Reset_PB);
_e2(CLK := gA[3].Input_DriveEnable);
_e3(CLK := gCmd_ResetPBGen);
TOF_0(IN := _e1.Q OR _e2.Q OR _e3.Q, PT := T#20ms);
gA[3].Cmd_Reset := TOF_0.Q;

(* Network 4: Cam Automat Synchronization Permissive *)
Synch_Permissive := NOT gA[3].Error AND gA[3].Ind_Homed AND gA[3].Ind_Enabled AND gA[9].Ind_Homed AND NOT gA[3].Ind_Homing;

(* Network 5: Cam Automat Synchronization Request *)
gA[3].Cmd_SynchronizedMotion := (NOT gA[3].Ind_AutomatEnabled OR gA[3].Cmd_SynchronizedMotion) AND Synch_Permissive AND NOT gRepeatChange;

(* Network 6: Conversion offset increment from mm/bag to inch/bag *)
rIncrOffsetAxeRun_Inch := gr_rIncrOffsetAxeRun / 25.4;

(* Network 7: Conversion offset increment from mm/bag to inch/bag *)
rIncrOffsetAxeRun_Inch := gr_rIncrOffsetAxeRun / 25.4;

(* Network 8: Advance Offset (+) *)
_e4(CLK := gA[4].Ind_bInContactZone);
IF g_bMachineRun AND gManualMode_On AND gA[3].Ind_SynchronizedMotion AND gI_SS_HoldingPos AND NOT gI_SS_HoldingNeg AND _e4.Q THEN
    gRecipeActive.Holding_Offset := gRecipeActive.Holding_Offset + rIncrOffsetAxeRun_Inch;
END_IF;

(* Network 9: Offset Retard (-) *)
_e5(CLK := gA[4].Ind_bInContactZone);
IF g_bMachineRun AND gManualMode_On AND gA[3].Ind_SynchronizedMotion AND gI_SS_HoldingNeg AND NOT gI_SS_HoldingPos AND _e5.Q THEN
    gRecipeActive.Holding_Offset := gRecipeActive.Holding_Offset + (rIncrOffsetAxeRun_Inch * -1.0);
END_IF;

(* Network 10: Limit The Offset To +/- The Active Repeat *)
gRecipeActive.Holding_Offset := LIMIT(MN := gRecipeActive.Repeat * -1.0, IN := gRecipeActive.Holding_Offset, MX := gRecipeActive.Repeat);

(* Network 11: Detect A Change and limit In Offset And Trigger A Relative Change In Phase Offset *)
H_FB_RelativeChangeLimitReal1_0(IN_bEnable := g_bMachineRun, IN_rMax := gr_rLimOffsetRunVal, IN_rMin := gr_rLimOffsetRunVal * -1.0, IN_rInput := 0.0, IN_rRepeat := gRecipeActive.Repeat, IN_rLimitIn := gRecipeActive.Holding_Offset);
IF H_FB_RelativeChangeLimitReal1_0.OUT_bChange AND gA[3].Ind_SynchronizedMotion THEN
    gA[3].Cmd_PhaseOffset := TRUE;
END_IF;
gA[3].SP_PhaseOffset := H_FB_RelativeChangeLimitReal1_0.OUT_rDiff;
gRecipeActive.Holding_Offset := H_FB_RelativeChangeLimitReal1_0.OUT_rLimitIn;

(* Network 12: Manu Axis motion timing setting (+) *)
gA[3].Cmd_ManuTimSetPlus := gManualMode_On AND NOT gA[9].Ind_InMotion AND NOT gMachine_Run AND NOT gMachine_Jog AND gI_SS_HoldingPos AND NOT gI_SS_HoldingNeg;

(* Network 13: Manu Axis motion timing setting (-) *)
gA[3].Cmd_ManuTimSetMinus := gManualMode_On AND NOT gA[9].Ind_InMotion AND NOT gMachine_Run AND NOT gMachine_Jog AND gI_SS_HoldingNeg AND NOT gI_SS_HoldingPos;
END_PROGRAM
```

### A3_Cycle.var
```iecst
(********************************************************************
 * COPYRIGHT -- .
 ********************************************************************
 * Program: A11_Cycle
 * File: A11_Cycle.var
 * Author: dominique
 * Created: August 01, 2011
 ********************************************************************
 * Local variables of program A11_Cycle
 ********************************************************************)

VAR
  iTest_          : ARRAY [0..9] OF INT ;
  rTempActPhasDeg : ARRAY[0..9] OF REAL ;
  rTempActOffsetInch : ARRAY[0..9] OF REAL ;
  rTemp_          : ARRAY[0..9] OF REAL ;
  stTON_01        : TON ;
END_VAR

VAR CONSTANT

END_VAR
```

### Program Logical/BagMachine_Section/Holding/Axis3/A3_Ref

#### A3_RefCyclic.ld
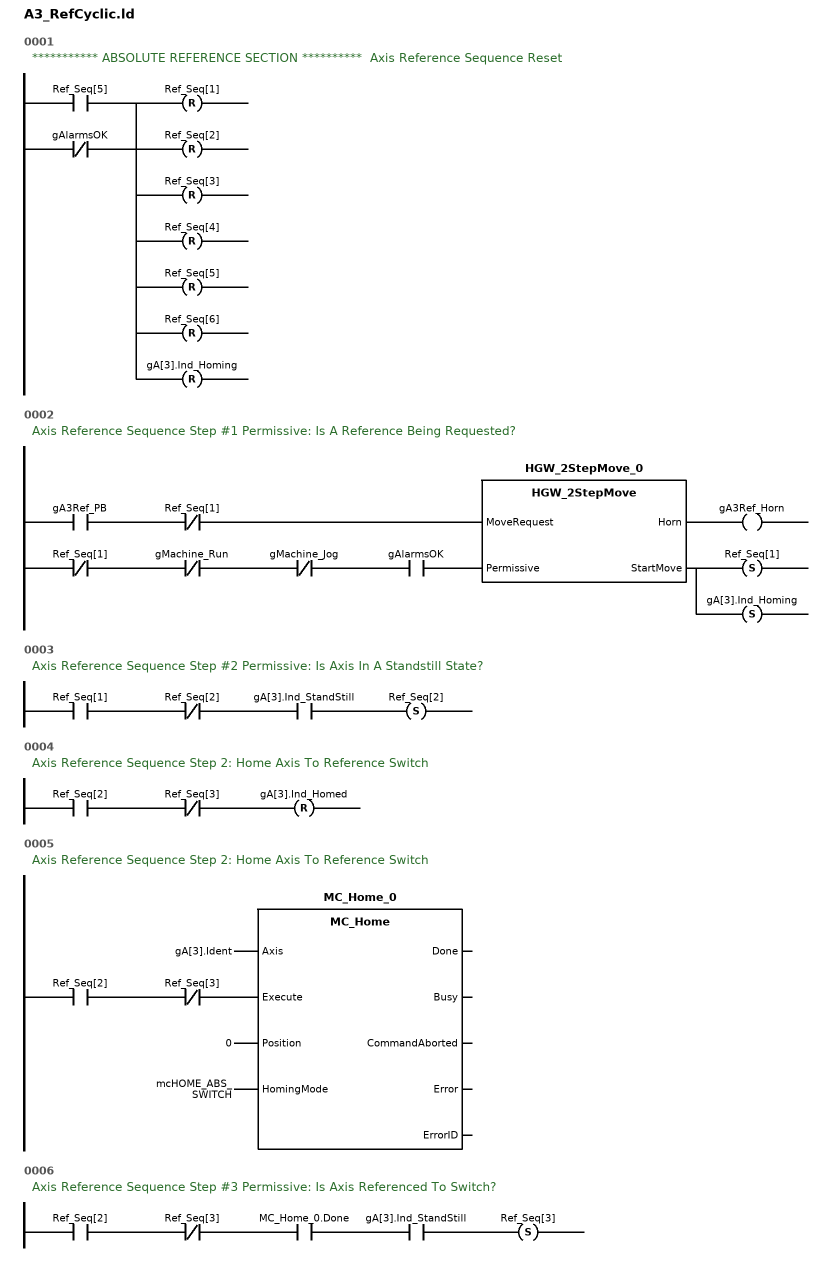
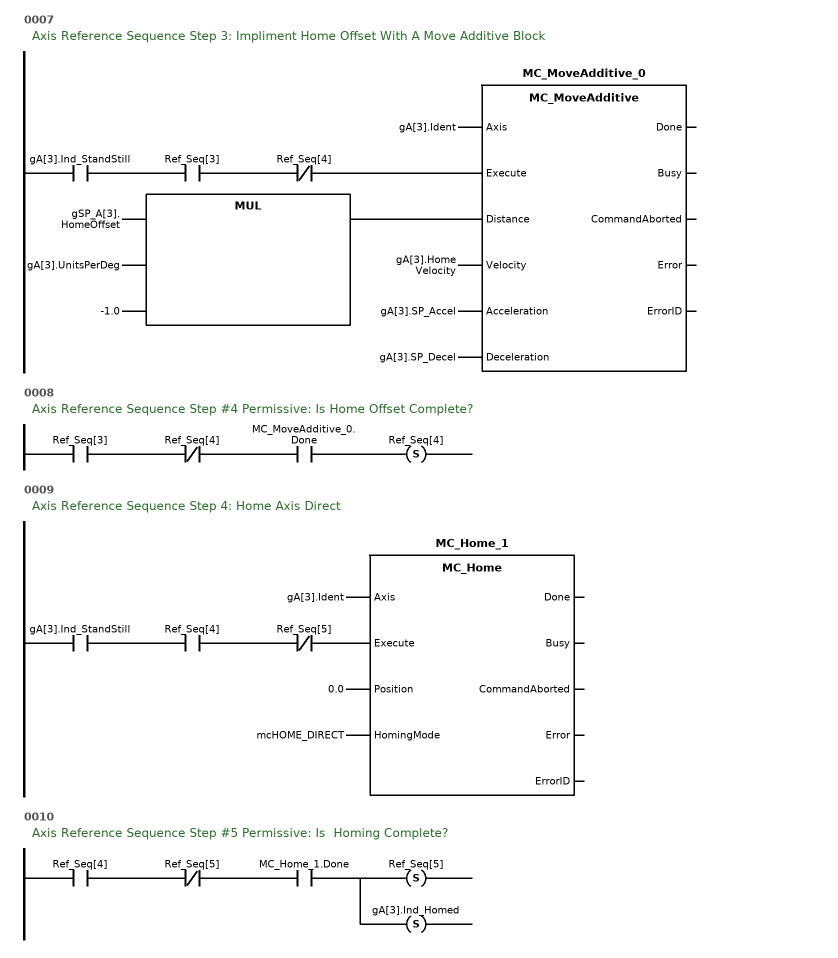
Ladder, written as Structured Text:
```iecst
(********************************************************************
 * COPYRIGHT -- Microsoft
 ********************************************************************
 * Program: A3_Ref
 * File: A3_RefCyclic.ld
 * Author: pkiel
 * Created: July 19, 2011
 ********************************************************************
 * Implementation of program A3_Ref
 ********************************************************************)

PROGRAM _CYCLIC
VAR
    _p1 : BOOL;
    _p2 : BOOL;
END_VAR
(* Network 1: *********** ABSOLUTE REFERENCE SECTION **********  Axis Reference Sequence Reset *)
_p1 := Ref_Seq[5];
IF Ref_Seq[5] OR NOT gAlarmsOK THEN Ref_Seq[1] := FALSE; END_IF;
IF _p1 OR NOT gAlarmsOK THEN
    Ref_Seq[2] := FALSE;
    Ref_Seq[3] := FALSE;
    Ref_Seq[4] := FALSE;
    Ref_Seq[5] := FALSE;
    Ref_Seq[6] := FALSE;
    gA[3].Ind_Homing := FALSE;
END_IF;

(* Network 2: Axis Reference Sequence Step #1 Permissive: Is A Reference Being Requested? *)
HGW_2StepMove_0(MoveRequest := gA3Ref_PB AND NOT Ref_Seq[1], Permissive := NOT Ref_Seq[1] AND NOT gMachine_Run AND NOT gMachine_Jog AND gAlarmsOK);
gA3Ref_Horn := HGW_2StepMove_0.Horn;
IF HGW_2StepMove_0.StartMove THEN
    Ref_Seq[1] := TRUE;
    gA[3].Ind_Homing := TRUE;
END_IF;

(* Network 3: Axis Reference Sequence Step #2 Permissive: Is Axis In A Standstill State? *)
IF Ref_Seq[1] AND NOT Ref_Seq[2] AND gA[3].Ind_StandStill THEN Ref_Seq[2] := TRUE; END_IF;

(* Network 4: Axis Reference Sequence Step 2: Home Axis To Reference Switch *)
IF Ref_Seq[2] AND NOT Ref_Seq[3] THEN gA[3].Ind_Homed := FALSE; END_IF;

(* Network 5: Axis Reference Sequence Step 2: Home Axis To Reference Switch *)
MC_Home_0(Axis := gA[3].Ident, Execute := Ref_Seq[2] AND NOT Ref_Seq[3], Position := 0, HomingMode := mcHOME_ABS_SWITCH);

(* Network 6: Axis Reference Sequence Step #3 Permissive: Is Axis Referenced To Switch? *)
IF Ref_Seq[2] AND NOT Ref_Seq[3] AND MC_Home_0.Done AND gA[3].Ind_StandStill THEN
    Ref_Seq[3] := TRUE;
END_IF;

(* Network 7: Axis Reference Sequence Step 3: Impliment Home Offset With A Move Additive Block *)
MC_MoveAdditive_0(Axis := gA[3].Ident, Execute := gA[3].Ind_StandStill AND Ref_Seq[3] AND NOT Ref_Seq[4], Distance := gSP_A[3].HomeOffset * gA[3].UnitsPerDeg * -1.0, Velocity := gA[3].HomeVelocity, Acceleration := gA[3].SP_Accel, Deceleration := gA[3].SP_Decel);

(* Network 8: Axis Reference Sequence Step #4 Permissive: Is Home Offset Complete? *)
IF Ref_Seq[3] AND NOT Ref_Seq[4] AND MC_MoveAdditive_0.Done THEN Ref_Seq[4] := TRUE; END_IF;

(* Network 9: Axis Reference Sequence Step 4: Home Axis Direct *)
MC_Home_1(Axis := gA[3].Ident, Execute := gA[3].Ind_StandStill AND Ref_Seq[4] AND NOT Ref_Seq[5], Position := 0.0, HomingMode := mcHOME_DIRECT);

(* Network 10: Axis Reference Sequence Step #5 Permissive: Is  Homing Complete? *)
_p2 := Ref_Seq[4] AND NOT Ref_Seq[5] AND MC_Home_1.Done;
IF Ref_Seq[4] AND NOT Ref_Seq[5] AND MC_Home_1.Done THEN Ref_Seq[5] := TRUE; END_IF;
IF _p2 THEN gA[3].Ind_Homed := TRUE; END_IF;
END_PROGRAM
```

### Program Logical/BagMachine_Section/HotGlue (IEC)

#### HotGlueCyclic.st - Cyclic code
```iecst
(********************************************************************
 * COPYRIGHT -- Microsoft
 ********************************************************************
 * Program: HotGlue
 * File: HotGlueCyclic.st
 * Author: pkiel
 * Created: July 14, 2011
 ********************************************************************
 * Implementation of program HotGlue
 ********************************************************************)

PROGRAM _CYCLIC

(* Glue Off/On From HMI *)
  HGW_2StatePB_0.PB := EDGEPOS(Glue_PB);
  GlueText_Ind := HGW_2StatePB_0.Text_Ind;
  GlueColor_Ind := HGW_2StatePB_0.Color_Ind;
  Glue_On := HGW_2StatePB_0.State1;
  HGW_2StatePB_0();

(* Glue Manual/Auto From HMI *)
	HGW_2StatePB_1.PB := (EDGEPOS(GlueAuto_PB) OR (NOT Glue_Auto AND gA[9].Ind_InMotion));
	GlueAutoText_Ind := HGW_2StatePB_1.Text_Ind;
	GlueAutoColor_Ind := HGW_2StatePB_1.Color_Ind;
	Glue_Auto := HGW_2StatePB_1.State1;
	HGW_2StatePB_1();

(* Glue Auto Pressure Based On Machine Speed *)
	HGW_ScaleReal_0.Enable := Glue_Auto;
	HGW_ScaleReal_0.InputMin := 0.0;
	HGW_ScaleReal_0.InputMax := 1000.0;
	HGW_ScaleReal_0.InputRaw := gActualMachineSpeed_FPM;
	HGW_ScaleReal_0.ScaledMin := LIMIT (0,gSP_HotGlue.MinPressure,400);
	HGW_ScaleReal_0.ScaledMax := LIMIT (0,gSP_HotGlue.MaxPressure,400);
	PressureCmd := HGW_ScaleReal_0.ScaledOut;
	HGW_ScaleReal_0();

(* Glue Manual Pressure *)
	IF (NOT Glue_Auto) THEN
		PressureCmd := gSP_HotGlue.ManPressure;
	END_IF

(* Glue Pressure Command Limit 0-100% *)
	PressureCmd := LIMIT (0,PressureCmd, 100);

(* If Disabled, Reduce Pressure To Zero *)
	IF (NOT Glue_On) THEN
		PressureCmd := 0;
	END_IF

(* Generate Analog Command To Seam Paste System Pressure *)
	HGW_ScaleReal_1.Enable := 1;
	HGW_ScaleReal_1.InputMin := 0.0;
	HGW_ScaleReal_1.InputMax := 100.0;
	HGW_ScaleReal_1.InputRaw := PressureCmd;
	HGW_ScaleReal_1.ScaledMin := 0.0;
	HGW_ScaleReal_1.ScaledMax := 32767.0;
	//gQ_CMD_HotGluePressure := REAL_TO_INT(HGW_ScaleReal_1.ScaledOut);
  gQ_CMD_UNW_GluePressure := REAL_TO_INT(HGW_ScaleReal_1.ScaledOut);
	HGW_ScaleReal_1();

(* Glue Auto On *)
	IF ((gActualMachineSpeed_BPM>=gSP_HotGlue.AutoOnSpeed) AND gA[9].Ind_InMotion AND Glue_On AND gBagMachine_WebBreakOK) THEN
		GlueAuto_On := 1;
	ELSE
		GlueAuto_On := 0;
	END_IF

(* Glue Gun Clean Control *)
	HGW_Toggle_0(In := GlueClean_PB , Time := T#12ms);

(* Glue Gun Control *)
	IF ((GlueAuto_On OR GluePurge_PB OR HGW_Toggle_0.Out) AND gAlarmsOK AND gI_SS_SeamGlueOnOff) THEN
		gQ_CR_HotGlue := 1;
	ELSE
		gQ_CR_HotGlue := 0;
	END_IF

(* Is 2nd Tube Selected *)
	IF (gSP_TubeSelect) THEN
		gQ_CR_HotGlueSelect := 1;
	ELSE
		gQ_CR_HotGlueSelect := 0;
  END_IF

END_PROGRAM
```

- Program Logical/BagMachine_Section/HotMicroPerf/Axis15/A15_Automat (IEC) (no source held here)

### Program Logical/BagMachine_Section/HotMicroPerf/Axis15/A15_Basic (IEC)

#### A15_BasicInit.st - Initialization code
```iecst
(********************************************************************
 * COPYRIGHT -- Microsoft
 ********************************************************************
 * Program: A15_Basic
 * File: A15_BasicInit.st
 * Author: dominique
 * Created: November 03, 2011
 ********************************************************************
 * Implementation of program A15_Basic
 ********************************************************************)

PROGRAM _INIT
	// Mecanical drive
  // Gear ratio = 48/20 x 48/25 x 48/48 = 24/5 x 48/25 = 576/125 = 4.608
	// Axis Setpoint Variables
		gA[15].SP_MotorPPR := 15625 / 2 ; // 36000 x 125 / 576  = 125 x 125 / 2 = 15625 / 2
		gA[15].SP_GearBoxInput:= 576;
		gA[15].SP_GearBoxOutput:= 125;
    gA[15].AxisPeriod := 36000 ; // D.M. 19/10/2011 B&H_14541  because of limited precsision  (gA[15].SP_MotorPPR*gA[15].SP_GearBoxInput/gA[15].SP_GearBoxOutput) = 35997.7 insted of 36000 and then the synchro is not correct
		gA[15].UnitsPerDeg := gA[15].AxisPeriod/360;
		gA[15].SP_Accel := 0.2*gA[15].AxisPeriod;
		gA[15].SP_Decel := 0.4*gA[15].AxisPeriod;
		gA[15].SP_EStopDecel := 1000.0*gA[15].AxisPeriod; // Stop axis from 1000 tr/min in 1s
    gA[15].HomeVelocity := 6*gA[15].AxisPeriod/60;
    gA[15].rSP_CorPosVel := 0.0 ;
    gA[15].rSP_OverrideV := 1.0 ;
    gA[15].rSP_OverrideA := 1.0 ;
    gA[15].Cmd_EStopDisable := 0 ;

	// access master axis
		AxisErrorNcAccess := ncaccess(ncACP10MAN, ADR('Axis15'), ADR(gA[15].Ident));

	// Trigger Initialization Of ModPosition
		InitModPosition:=1;

END_PROGRAM
```

### A15_Control.var
```iecst
(********************************************************************
 * COPYRIGHT -- Microsoft
 ********************************************************************
 * Program: A15_Control
 * File: A15_Control.var
 * Author: dominique
 * Created: November 03, 2011
 ********************************************************************
 * Local variables of program A15_Control
 ********************************************************************)
VAR
	HGW_ChangeReal_0 : HGW_ChangeReal;
	HGW_RelativeChangeReal_0 : H_FB_RelativeChangeLimitReal1;
	HGW_Toggle_0 : HGW_Toggle;
	Synch_Permissive : BOOL;
	TOF_0 : TOF;
	TON_0 : TON;
  rIncrOffsetAxeRun_Inch : REAL ;

  bToolSizeChange : BOOL ;
END_VAR
```

### Program Logical/BagMachine_Section/HotMicroPerf/Axis15/A15_Cycle

#### A15_CycleCyclic.st
```iecst
(********************************************************************
 * COPYRIGHT -- .
 ********************************************************************
 * Program: A15_Cycle
 * File: A15_CycleCyclic.st
 * Author: dominique
 * Created: November 03, 2011
 ********************************************************************
 * Implementation of program A15_Cycle
 ********************************************************************)

PROGRAM _CYCLIC

// Manu axis movement for timing setting

    //---------------------------------------------------------------------------------------------------------------------
    // Timing setting cycle
    //---------------------------------------------------------------------------------------------------------------------
    // Start cycle
    gstCycA[15].CycManTimSet.CmdStart := ( gA[15].Cmd_ManuTimSetPlus    OR
                                           gA[15].Cmd_ManuTimSetMinus ) AND
                                         gA[15].Ind_Ready                ;
    IF gstCycA[15].CycManTimSet.CmdStart THEN
      gstCycA[15].CycManTimSet.bSCyc := 1 ;
    END_IF ;

    //----------------------------------------------------------------------
    // Cycle at rest
    IF NOT(gstCycA[15].CycManTimSet.bSCyc) AND
       1                                 THEN
      IF NOT( gstCycA[15].CycManTimSet.bFCyc ) THEN
        // Init after cycle unpropaly ended
        gstCycA[15].CycManTimSet.bFCyc := 1 ;
        gstCycA[15].CycManTimSet.bCyc  := 0 ;

        gstCycA[15].CycManTimSet.CmdMov       := 0 ;
        gstCycA[15].CycManTimSet.CmdStop      := 0 ;
        gstCycA[15].CycManTimSet.CmdSynchroOn := 0 ;
      END_IF
      gstCycA[15].CycManTimSet.iStep := 0 ;
      RETURN ;
    ELSE
    //----------------------------------------------------------------------
    // Cycle running

      // Permanent conditions
      IF NOT(gA[15].Ind_Ready)                  OR
         NOT(gstCycA[15].CycManTimSet.CmdStart) AND
         (gstCycA[15].CycManTimSet.iStep <= 2)  THEN
        gstCycA[15].CycManTimSet.bSCyc := 0 ;
        RETURN ;
      END_IF

      // Permanent actions
      stTON_01 (
            IN := ( gstCycA[15].CycManTimSet.iStep = C_iSTEP_0 ) ,
            PT := T#30ms
               ) ;
    END_IF
    //----------------------------------------------------------------------
    // Cycle steps

        CASE gstCycA[15].CycManTimSet.iStep OF

        C_iSTEP_0 :
         //----------------------------------------------
         // Step 1 : Initialisation
         //----------------------------------------------
          IF stTON_01.Q THEN
            gstCycA[15].CycManTimSet.iStep := C_iSTEP_1 ;

            // Action Step 1
            gstCycA[15].CycManTimSet.bFCyc := 0 ;
            gstCycA[15].CycManTimSet.bCyc  := 1 ;
          END_IF

        C_iSTEP_1 :
         //----------------------------------------------
         // Step 2 : Synchro Drum
         //----------------------------------------------
          IF TRUE THEN
            gstCycA[15].CycManTimSet.iStep := C_iSTEP_2 ;

            // Action Step 2
            gstCycA[15].CycManTimSet.CmdSynchroOn := 1 ;
          END_IF

        C_iSTEP_2 :
         //----------------------------------------------
         // Step 3 : Activation motion and Stop waiting
         //----------------------------------------------
          IF gstCycA[15].CycManTimSet.bSynchroOkSlavA[7] THEN
            gstCycA[15].CycManTimSet.iStep := C_iSTEP_3 ;

            // Action Step 3
            gstCycA[15].CycManTimSet.CmdMov  := 1 ;
            gstCycA[15].CycManTimSet.CmdStop := 0 ;
            // Stop waiting
          END_IF

        C_iSTEP_3 :
         //----------------------------------------------
         // Step 4 : Stop motion and End stop waiting
         //----------------------------------------------
          IF NOT(gstCycA[15].CycManTimSet.CmdStart) THEN
            gstCycA[15].CycManTimSet.iStep := C_iSTEP_4 ;

            // Action Step 4
            gstCycA[15].CycManTimSet.CmdMov  := 0 ;
            gstCycA[15].CycManTimSet.CmdStop := 1 ;
            // End stop waiting
          END_IF

        C_iSTEP_4 :
         //----------------------------------------------
         // Step 3 : Activation motion and Stop waiting
         // Step 5 : Cut synchro
         //----------------------------------------------
          // Condition Step3
          IF gstCycA[15].CycManTimSet.CmdStart THEN
            gstCycA[15].CycManTimSet.iStep := C_iSTEP_3 ;

            // Action Step 3
            gstCycA[15].CycManTimSet.CmdMov  := 1 ;
            gstCycA[15].CycManTimSet.CmdStop := 0 ;
            // Stop waiting
            RETURN ;
          END_IF ;
          // Condition Step5
          IF NOT(gstCycA[15].CycManTimSet.CmdStop) THEN
            gstCycA[15].CycManTimSet.iStep := C_iSTEP_5 ;

            // Action Step 5
            gstCycA[15].CycManTimSet.CmdSynchroOn := 0 ;
          END_IF

        C_iSTEP_5 :
         //----------------------------------------------
         // Step 6 : New offset calculation
         //----------------------------------------------
          IF TRUE THEN
            gstCycA[15].CycManTimSet.iStep := C_iSTEP_6 ;

            // Action Step 6
            // Memo Actual phase Offset
            rTempActPhasDeg[7]    := gRecipeActive.rDrum_PhasMasterDeg ;
            rTempActOffsetInch[7] := gRecipeActive.Drum_Offset ;
            // Update phase
            gRecipeActive.rDrum_PhasMasterDeg := gA[15].rActPhasDeg ;
            // Update Offset
            rTemp_[7] := rTempActOffsetInch[7] + (gRecipeActive.rDrum_PhasMasterDeg - rTempActPhasDeg[7])*gA[15].InchPerDeg ;
            gRecipeActive.Drum_Offset := H_FC_Modulus (IN_rMod := gRecipeActive.Repeat, IN_rVar := rTemp_[7]) ;
          END_IF

        C_iSTEP_6 :
         //----------------------------------------------
         // Step 0 : First step
         //----------------------------------------------
          IF TRUE THEN
            gstCycA[15].CycManTimSet.iStep := C_iSTEP_0 ;

            // Action Step 0
            gstCycA[15].CycManTimSet.bSCyc := 0 ;
            gstCycA[15].CycManTimSet.bFCyc := 1 ;
            gstCycA[15].CycManTimSet.bCyc  := 0 ;
          END_IF
        END_CASE
    //---------------------------------------------------------------------------------------------------------------------

END_PROGRAM
```

#### A15_CycleInit.st
```iecst
(********************************************************************
 * COPYRIGHT -- .
 ********************************************************************
 * Program: A15_Cycle
 * File: A15_CycleInit.st
 * Author: dominique
 * Created: November 03, 2011
 ********************************************************************
 * Implementation of program A15_Cycle
 ********************************************************************)

PROGRAM _INIT

END_PROGRAM
```

### Data object Logical/BagMachine_Section/HotMicroPerf/Axis15/A15_Init (Ax)

#### A15_Init.ax
```
InitParameter (Version=2.21.1, NcSwId=ACP10)
  ACP10AXIS_typ:
    dig_in:
      level:
        reference = ncACTIV_HI
        pos_hw_end = ncACTIV_HI
        neg_hw_end = ncACTIV_HI
        trigger1 = ncACTIV_HI
        trigger2 = ncACTIV_HI
    encoder_if:
      parameter:
        count_dir = ncINVERSE
        scaling:
          load:
            units = 15625
            rev_motor = 2
    limit:
      parameter:
        v_pos = 600000.0
        v_neg = 600000.0
        a1_pos = 5e+006
        a2_pos = 5e+006
        a1_neg = 5e+006
        a2_neg = 5e+006
        t_jolt = 0.1
        t_in_pos = 0.5
        pos_sw_end = 8388607
        neg_sw_end = -8388608
        ds_warning = 500.0
        ds_stop = 1000.0
        a_stop = 1e+030
        dv_stop = 0
        dv_stop_mode = ncOFF
    controller:
      mode = ncPOSITION
      position:
        kv = 30.0
        tn = 0.0
        t_predict = 0.0004
        t_total = 0.0012
        p_max = 1e+030
        i_max = 0.0
      speed:
        kv = 4.0
        tn = 0.0
        t_filter = 0.0
        isq_filter1:
          type = ncOFF
          a0 = 0.0
          a1 = 0.0
          b0 = 0.0
          b1 = 0.0
          b2 = 0.0
          c0_par_id = 0
          c1_par_id = 0
        isq_filter2:
          type = ncOFF
          a0 = 0.0
          a1 = 0.0
          b0 = 0.0
          b1 = 0.0
          b2 = 0.0
          c0_par_id = 0
          c1_par_id = 0
        isq_filter3:
          type = ncOFF
          a0 = 0.0
          a1 = 0.0
          b0 = 0.0
          b1 = 0.0
          b2 = 0.0
          c0_par_id = 0
          c1_par_id = 0
      uf:
        type = ncLINEAR
        auto_config = ncMOTOR_PAR
        u0 = 0.0
        un = 0.0
        fn = 50.0
        k_f_slip = 0.0
      ff:
        torque_load = 0.0
        torque_pos = 0.0
        torque_neg = 0.0
        kv_torque = 0.0
        inertia = 0.0
        t_filter_a = 0.0
    move:
      stop:
        parameter[0]:
          decel_ramp = ncA_LIMIT
          controller = ncON
        parameter[1]:
          decel_ramp = ncA_LIMIT
          controller = ncON
        parameter[2]:
          decel_ramp = ncA_LIMIT
          controller = ncON
        parameter[3]:
          decel_ramp = ncA_LIMIT
          controller = ncON
        quickstop:
          decel_ramp = ncA_LIMIT
        drive_error:
          decel_ramp = ncA_LIMIT
      homing:
        parameter:
          s = 0
          v_switch = 3600.0
          v_trigger = 360.0
          a = 50000.0
          mode = ncHOME_OFFSET
          edge_sw = ncPOSITIVE
          start_dir = ncPOSITIVE
          trigg_dir = ncPOSITIVE
          ref_pulse = ncOFF
          tr_s_block = 0.0
      basis:
        parameter:
          v_pos = 36000.0
          v_neg = 100000.0
          a1_pos = 50000.0
          a2_pos = 50000.0
          a1_neg = 50000.0
          a2_neg = 50000.0
    message:
      text:
        parameter:
          format = ncBREAK
          columns = 80
          data_modul = Error_Eng
```

### Program Logical/BagMachine_Section/HotMicroPerf/Axis15/A15_MotionCycle (IEC)

#### A15_MotionCycleInit.st - Initialization code
```iecst
(********************************************************************
 * COPYRIGHT -- .
 ********************************************************************
 * Program: A15_MotionCycle
 * File: A15_MotionCycleInit.st
 * Author: dominique
 * Created: November 06, 2011
 ********************************************************************
 * Implementation of program A15_MotionCycle
 ********************************************************************)

PROGRAM _INIT

  rTest := 0 ;

END_PROGRAM
```

#### A15_MotionCycle.var - Local variables
```iecst
(********************************************************************
 * COPYRIGHT -- .
 ********************************************************************
 * Program: A15_MotionCycle
 * File: A15_MotionCycle.var
 * Author: dominique
 * Created: November 03, 2011
 ********************************************************************
 * Local variables of program A15_MotionCycle
 ********************************************************************)

VAR

  bQ_SOL_HMP_BrushForward : BOOL ;
  bQ_SOL_HMP_ProtecDown   : BOOL ;
  rLS_Act_mmin            : REAL ;
  rTest  : REAL ;
  rTest1 : REAL ;
  bTest  : BOOL ;
  rCalc  : ARRAY[0..9] OF REAL ;

  stTON_0 : TON ;
  stTON_1 : TON ;
  MC_CamIn_0  : MC_CamIn ;
  uiMC_CamIn_ErrorID : UINT ;
  MC_GearIn_0 : MC_GearIn ;
  uiMC_GearIn_ErrorID : UINT ;
  MC_GearOut_0 : MC_GearOut ;
  uiMC_GearOut_ErrorID : UINT ;
  bGearInError : BOOL ;

END_VAR

VAR CONSTANT

END_VAR
```

### Program Logical/BagMachine_Section/HotMicroPerf/Axis15/A15_Ref

#### A15_Ref.var
```iecst
(********************************************************************
 * COPYRIGHT -- Microsoft
 ********************************************************************
 * Program: A15_Ref
 * File: A15_Ref.var
 * Author: dominique
 * Created: November 03, 2011
 ********************************************************************
 * Local variables of program A15_Ref
 ********************************************************************)
VAR
	HGW_2StepMove_0 : HGW_2StepMove;
	MC_Home_0 : MC_Home;
	MC_Home_1 : MC_Home;
	MC_MoveAdditive_0 : MC_MoveAdditive;
	Ref_Seq : ARRAY[0..10] OF BOOL;
END_VAR
```

#### A15_RefCyclic.ld
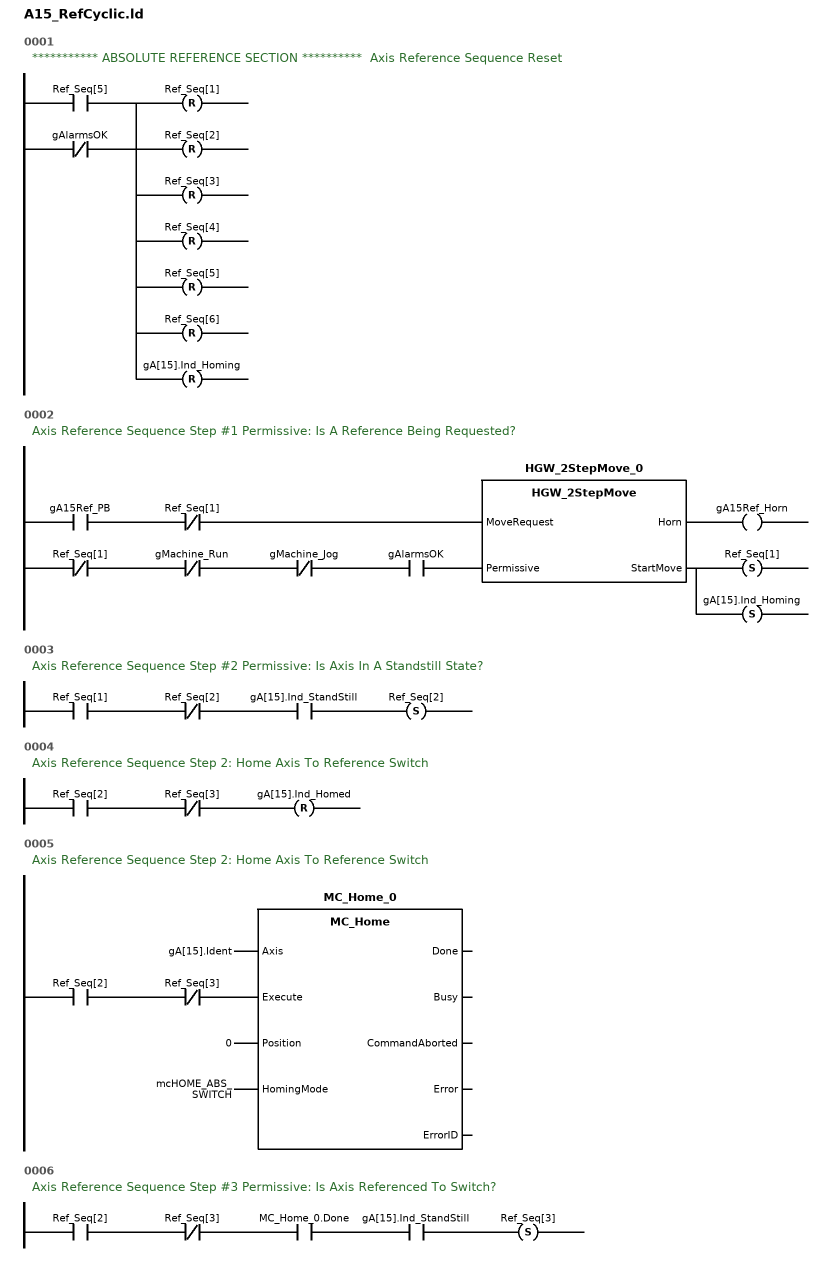
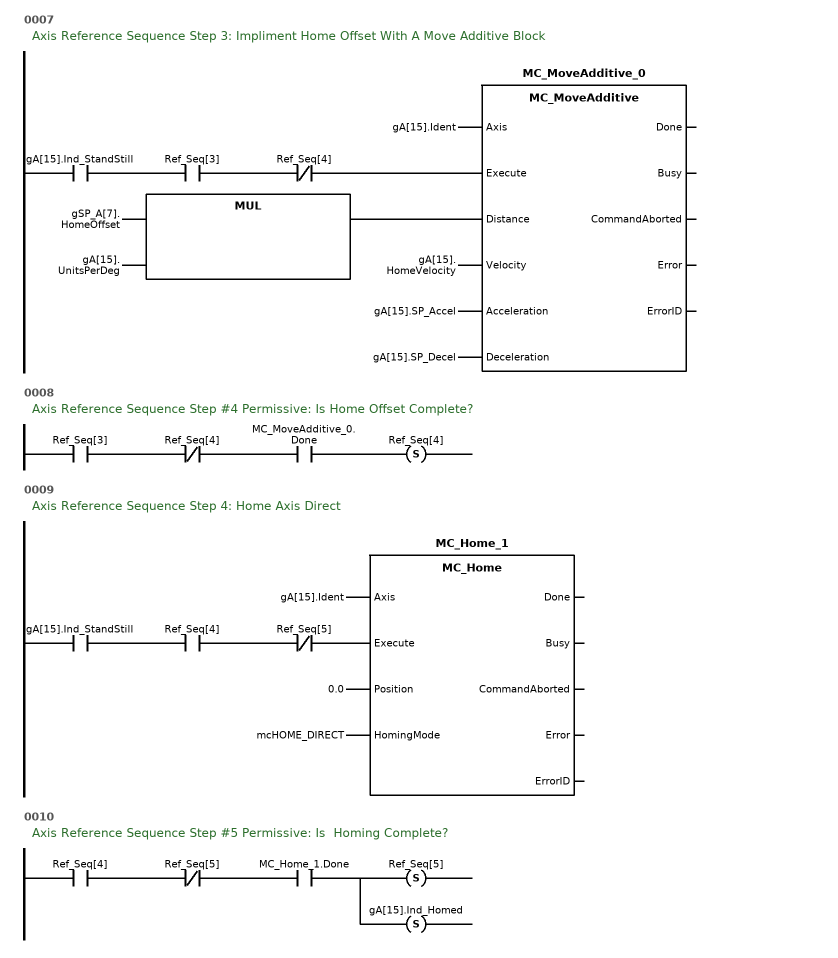
Ladder, written as Structured Text:
```iecst
(********************************************************************
 * COPYRIGHT -- Microsoft
 ********************************************************************
 * Program: A7_Ref
 * File: A7_RefCyclic.ld
 * Author: pkiel
 * Created: July 19, 2011
 ********************************************************************
 * Implementation of program A7_Ref
 ********************************************************************)

PROGRAM _CYCLIC
VAR
    _p1 : BOOL;
    _p2 : BOOL;
END_VAR
(* Network 1: *********** ABSOLUTE REFERENCE SECTION **********  Axis Reference Sequence Reset *)
_p1 := Ref_Seq[5];
IF Ref_Seq[5] OR NOT gAlarmsOK THEN Ref_Seq[1] := FALSE; END_IF;
IF _p1 OR NOT gAlarmsOK THEN
    Ref_Seq[2] := FALSE;
    Ref_Seq[3] := FALSE;
    Ref_Seq[4] := FALSE;
    Ref_Seq[5] := FALSE;
    Ref_Seq[6] := FALSE;
    gA[15].Ind_Homing := FALSE;
END_IF;

(* Network 2: Axis Reference Sequence Step #1 Permissive: Is A Reference Being Requested? *)
HGW_2StepMove_0(MoveRequest := gA15Ref_PB AND NOT Ref_Seq[1], Permissive := NOT Ref_Seq[1] AND NOT gMachine_Run AND NOT gMachine_Jog AND gAlarmsOK);
gA15Ref_Horn := HGW_2StepMove_0.Horn;
IF HGW_2StepMove_0.StartMove THEN
    Ref_Seq[1] := TRUE;
    gA[15].Ind_Homing := TRUE;
END_IF;

(* Network 3: Axis Reference Sequence Step #2 Permissive: Is Axis In A Standstill State? *)
IF Ref_Seq[1] AND NOT Ref_Seq[2] AND gA[15].Ind_StandStill THEN Ref_Seq[2] := TRUE; END_IF;

(* Network 4: Axis Reference Sequence Step 2: Home Axis To Reference Switch *)
IF Ref_Seq[2] AND NOT Ref_Seq[3] THEN gA[15].Ind_Homed := FALSE; END_IF;

(* Network 5: Axis Reference Sequence Step 2: Home Axis To Reference Switch *)
MC_Home_0(Axis := gA[15].Ident, Execute := Ref_Seq[2] AND NOT Ref_Seq[3], Position := 0, HomingMode := mcHOME_ABS_SWITCH);

(* Network 6: Axis Reference Sequence Step #3 Permissive: Is Axis Referenced To Switch? *)
IF Ref_Seq[2] AND NOT Ref_Seq[3] AND MC_Home_0.Done AND gA[15].Ind_StandStill THEN
    Ref_Seq[3] := TRUE;
END_IF;

(* Network 7: Axis Reference Sequence Step 3: Impliment Home Offset With A Move Additive Block *)
MC_MoveAdditive_0(Axis := gA[15].Ident, Execute := gA[15].Ind_StandStill AND Ref_Seq[3] AND NOT Ref_Seq[4], Distance := gSP_A[7].HomeOffset * gA[15].UnitsPerDeg, Velocity := gA[15].HomeVelocity, Acceleration := gA[15].SP_Accel, Deceleration := gA[15].SP_Decel);

(* Network 8: Axis Reference Sequence Step #4 Permissive: Is Home Offset Complete? *)
IF Ref_Seq[3] AND NOT Ref_Seq[4] AND MC_MoveAdditive_0.Done THEN Ref_Seq[4] := TRUE; END_IF;

(* Network 9: Axis Reference Sequence Step 4: Home Axis Direct *)
MC_Home_1(Axis := gA[15].Ident, Execute := gA[15].Ind_StandStill AND Ref_Seq[4] AND NOT Ref_Seq[5], Position := 0.0, HomingMode := mcHOME_DIRECT);

(* Network 10: Axis Reference Sequence Step #5 Permissive: Is  Homing Complete? *)
_p2 := Ref_Seq[4] AND NOT Ref_Seq[5] AND MC_Home_1.Done;
IF Ref_Seq[4] AND NOT Ref_Seq[5] AND MC_Home_1.Done THEN Ref_Seq[5] := TRUE; END_IF;
IF _p2 THEN gA[15].Ind_Homed := TRUE; END_IF;
END_PROGRAM
```

### Program Logical/BagMachine_Section/HotMicroPerf/HMPerf_Gen

#### HMPerf_Gen.var
```iecst
(********************************************************************
 * COPYRIGHT -- .
 ********************************************************************
 * Program: HMPerf_Gen
 * File: HMPerf_Gen.var
 * Author: dominique
 * Created: November 05, 2011
 ********************************************************************
 * Local variables of program HMPerf_Gen
 ********************************************************************)

VAR CONSTANT

END_VAR

VAR
  HMI_HMPerf_bModePB : BOOL ; (*Operation mode =0:Continu, =1:Interrupt*)

  bInterruptReq : BOOL;
  bContinuReq   : BOOL;
  bOnReq        : BOOL;
  bOffReq       : BOOL;
  bOn_PB        : BOOL ;
  bOff_PB       : BOOL ;

  bToolSizeLock : BOOL ;
  bToolUpLock   : BOOL ;
  bOffsetLock   : BOOL ;
  iToolUpVisibl : INT ;
  bReadyInd     : BOOL;

  iOperState         : INT ; (*Operation State, =0:Off, =1:Slow Rotation, =2:Synchronized, =3:Fault*)
  uiOperStateCol_Ind : UINT ;
  iHeatState         : INT ; (*Heater State, =0:Off, =1:On, =2:/, =3:Fault*)
  uiHeatStateCol_Ind : UINT ;

  stTOF_0 : TOF ;
  bQ_CR_DRY_Blower      : BOOL;
  bQ_CR_DRY_HeatRegul   : BOOL;
  bQ_CR_DRY_HeatContinu : BOOL;
END_VAR

VAR RETAIN
  HGW_2StatePB_0 : HGW_2StatePB;
END_VAR
```

#### HMPerf_GenInit.st
```iecst
(********************************************************************
 * COPYRIGHT -- .
 ********************************************************************
 * Program: HMPerf_Gen
 * File: HMPerf_GenInit.st
 * Author: dominique
 * Created: November 05, 2011
 ********************************************************************
 * Implementation of program HMPerf_Gen
 ********************************************************************)

PROGRAM _INIT

  // Printing Manual/Auto PB Colors
  HGW_2StatePB_0.BackColor_State0 := gYellow;
  HGW_2StatePB_0.ForeColor_State0 := gBlack;
  HGW_2StatePB_0.BackColor_State1 := gGreen;
  HGW_2StatePB_0.ForeColor_State1 := gBlack;

  HMI_HMPerf_bModePB := gRecipeActive.bHMPerf_Mode ;

END_PROGRAM
```

### Data object Logical/BagMachine_Section/MasterAxis/A9_Init/A9_Init (Vax) - ACP10: Virtual Axis data object.

- A9_Init.vax (not shown)

### Program Logical/BagMachine_Section/MasterAxis/A9_Init/A9_Basic (IEC) - Basic Servo

#### A9_BasicCyclic.st - Cyclic code
```iecst
(********************************************************************
 * COPYRIGHT -- Microsoft
 ********************************************************************
 * Program: A9_Basic
 * File: A9_BasicCyclic.st
 * Author: pkiel
 * Created: July 12, 2011
 ********************************************************************
 * Implementation of program A9_Basic
 ********************************************************************)

PROGRAM _CYCLIC

	gA[9].UnitsPerInch := gA[9].AxisPeriod/gRecipeActive.Repeat;

	IF (gA[9].Ident<>0) THEN

	(************************ READ DRIVE STATUS *************************)
	(* Access to the following bools:
	gA[x]_DriveStatus.Simulation			: If TRUE, simulation mode is active
	gA[x]_DriveStatus.NetworkInit			: If TRUE, the network is initialized
	gA[x]_DriveStatus.HomeSwitch			: If TRUE, the digital reference switch input is active
	gA[x]_DriveStatus.PosHWSwitch			: If TRUE, the positive hardware end switch is active
	gA[x]_DriveStatus.NegHWSwitch			: If TRUE, the negative hardware end switch is active
	gA[x]_DriveStatus.Trigger1				: If TRUE, the first trigger input is active
	gA[x]_DriveStatus.Trigger2				: If TRUE, the second trigger input is active
	gA[x]_DriveStatus.DriveEnable			: If TRUE, the enable input is active
	gA[x]_DriveStatus.ControllerReady		: If TRUE, the controller is ready to beturned on
	gA[x]_DriveStatus.ControllerStatus		: If TRUE, the controller is turned on (Same as MC_Power.Status)
	gA[x]_DriveStatus.AxisError				: If TRUE, at least one error has occurred (not acknowledged)
	gA[x]_DriveStatus.LagWarning			: If TRUE, the lag error has exceeded the limit value specified for a warning*)
		MC_BR_ReadDriveStatus_0.Enable := 1;
		MC_BR_ReadDriveStatus_0.Axis := gA[9].Ident;
		MC_BR_ReadDriveStatus_0.AdrDriveStatus := ADR (DriveStatus);
		MC_BR_ReadDriveStatus_0();
		gA[9].Ind_Simulation		:=	DriveStatus.Simulation;
		gA[9].Ind_NetworkInit		:=	DriveStatus.NetworkInit;
		gA[9].Input_Home			:=	DriveStatus.HomeSwitch;
		gA[9].Input_PosHW			:=	DriveStatus.PosHWSwitch;
		gA[9].Input_NegHW			:=	DriveStatus.NegHWSwitch;
		gA[9].Input_Trigger1		:=	DriveStatus.Trigger1;
		gA[9].Input_Trigger2		:=	DriveStatus.Trigger2;
		gA[9].Input_DriveEnable		:=	DriveStatus.DriveEnable;
		gA[9].Ind_ControllerReady	:=	DriveStatus.ControllerReady;
		gA[9].Ind_ControllerStatus	:=	DriveStatus.ControllerStatus;
		gA[9].Error					:=	DriveStatus.AxisError;
		gA[9].Ind_LagWarning		:=	DriveStatus.LagWarning;

	(************************ READ AXIS ERROR **********************)
		MC_ReadAxisError_0.Enable := gA[9].Ind_NetworkInit;
		MC_ReadAxisError_0.Axis := gA[9].Ident;
		MC_ReadAxisError_0.DataAddress := ADR(gA[9].ErrorText);
		MC_ReadAxisError_0.DataLength := SIZEOF(gA[9].ErrorText);
		MC_ReadAxisError_0.DataObjectName := 'Error_Eng';
		MC_ReadAxisError_0();
		IF(MC_ReadAxisError_0.Valid) THEN
			gA[9].ErrorID := MC_ReadAxisError_0.AxisErrorID;
			gA[9].ErrorCount := MC_ReadAxisError_0.AxisErrorCount;
		END_IF
	(* Auto Acknowledge Errors *)
		IF (gA[9].Cmd_Reset AND (gA[9].ErrorCount<>0) AND NOT AutoAck) THEN
			AutoAck:=1;
		ELSE
			AutoAck:=0;
		END_IF
	(*Axis Error Acknowledge*)
		IF (EDGEPOS(AutoAck) OR EDGEPOS(gA[9].ErrorAck)) THEN
			MC_ReadAxisError_0.Acknowledge := 1;
		ELSE;
			MC_ReadAxisError_0.Acknowledge :=0;
		END_IF

	(************************ RESET AXIS ERROR **********************)
		IF (gA[9].Cmd_Reset AND (gA[9].ErrorCount=0) AND gA[9].ErrorStop) THEN
			MC_Reset_0.Execute:=1;
		END_IF
		IF (MC_Reset_0.Done) THEN
			MC_Reset_0.Execute:=0;
			gA[9].Cmd_Reset:=0;
			ResetError := 0;
		END_IF
		IF (MC_Reset_0.Error) THEN
			MC_Reset_0.Execute:=0;
			gA[9].Cmd_Reset:=0;
			ResetError := 1;
		END_IF
		MC_Reset_0.Axis:=gA[9].Ident;
		MC_Reset_0();

	(************************ READ AXIS STATUS *************************)
		MC_ReadStatus_0.Enable := gA[9].Ind_NetworkInit;
		MC_ReadStatus_0.Axis := gA[9].Ident;
		MC_ReadStatus_0();
		IF(MC_ReadStatus_0.Valid = TRUE)THEN
			gA[9].Ind_Enabled 			:= NOT (MC_ReadStatus_0.Disabled);
			gA[9].Ind_StandStill		:= MC_ReadStatus_0.StandStill;
			gA[9].Ind_Stopping			:= MC_ReadStatus_0.Stopping;
			gA[9].Ind_DiscreteMotion	:= MC_ReadStatus_0.DiscreteMotion;
			gA[9].Ind_ContinuousMotion	:= MC_ReadStatus_0.ContinuousMotion;
			gA[9].Ind_SynchronizedMotion:= MC_ReadStatus_0.SynchronizedMotion;
			gA[9].ErrorStop				:= MC_ReadStatus_0.Errorstop;
		END_IF

	(******************** INIT POSITION MODULUS  *********************)
		MC_BR_InitModPos_0.Execute:= InitModPosition;
		MC_BR_InitModPos_0.Axis:= gA[9].Ident;
		MC_BR_InitModPos_0.Period:= REAL_TO_UDINT(gA[9].AxisPeriod);
		MC_BR_InitModPos_0.Factor:=1;
		InitModPos_Done:=MC_BR_InitModPos_0.Done;
		MC_BR_InitModPos_0();

	(******************** INIT ENDLESS POSITION *********************)
		MC_BR_InitEndlessPosition_0.Execute:= InitModPos_Done;
		MC_BR_InitEndlessPosition_0.Axis:= gA[9].Ident;
		MC_BR_InitEndlessPosition_0.DataAddress:= ADR(gEndPosData[9]);
		IF (MC_BR_InitEndlessPosition_0.Done) THEN
			InitModPosition:=0;
			InitEndlessPosition:=0;
			HomeRestore:=1;
		END_IF
		MC_BR_InitEndlessPosition_0();
    stTON_0(IN:=HomeRestore, PT:=T#5s) ;

	(************************ HOME AXIS FIRST POWER UP **********************)
		IF (HomeRestore AND NOT gA9_FirstHomed) AND
       stTON_0.Q                            AND
       ( gA[9].Ind_StandStill               OR
         NOT(gA[9].Ind_Enabled ) )          THEN
			MC_Home_0.Execute:= 1 ;
		END_IF
		MC_Home_0.Axis:=gA[9].Ident;
		MC_Home_0.Position:=0;
		MC_Home_0.HomingMode:=mcHOME_DIRECT;
		IF (MC_Home_0.Done) THEN
			MC_Home_0.Execute:=0;
			gA9_FirstHomed:=1;
		END_IF
		MC_Home_0();
    stTON_1(IN:=gA9_FirstHomed, PT:=T#5s) ;

	(************************ HOME AXIS **********************)
    IF (gA9_FirstHomed AND stTON_1.Q) AND
       ( gA[9].Ind_StandStill         OR
         NOT(gA[9].Ind_Enabled ) )    THEN
      MC_Home_1.Execute:=HomeRestore ;
		END_IF
		MC_Home_1.Axis:=gA[9].Ident;
		MC_Home_1.Position:=0;
		MC_Home_1.HomingMode:=mcHOME_RESTORE_POS;
		IF (MC_Home_1.Done) THEN
			gA[9].Ind_Homed:=1;
			HomeRestore:=0;
		END_IF
		MC_Home_1();

	(******************** READ ACTUAL POSITION *********************)
		MC_ReadActualPosition_0.Enable:= gA[9].Ind_NetworkInit;
		MC_ReadActualPosition_0.Axis:= gA[9].Ident;
		MC_ReadActualPosition_0();
		IF(MC_ReadActualPosition_0.Valid = TRUE)THEN
			gA[9].PositionCount := MC_ReadActualPosition_0.Position;
			gA[9].PositionInch := gA[9].PositionCount/gA[9].UnitsPerInch;
			gA[9].PositionDeg := gA[9].PositionCount/gA[9].UnitsPerDeg;
		END_IF

	(******************** READ ACTUAL VELOCITY *********************)
		IF(MC_ReadActualVelocity_0.Error=TRUE) THEN
			MC_ReadActualVelocity_0.Enable:= 0;
		ELSE
			MC_ReadActualVelocity_0.Enable:= 1;
		END_IF
		MC_ReadActualVelocity_0.Axis:= gA[9].Ident;
		MC_ReadActualVelocity_0();
		IF(MC_ReadActualVelocity_0.Valid = TRUE)THEN
			gA[9].ActualVelocity := MC_ReadActualVelocity_0.Velocity*60/gA[9].SP_MotorPPR;
			IF (gA[9].ActualVelocity>1) THEN
				gA[9].Ind_InMotion:=1;
			ELSE
				gA[9].Ind_InMotion:=0;
			END_IF
		END_IF

		gActualMachineSpeed_BPM := MC_ReadActualVelocity_0.Velocity*60/gA[9].AxisPeriod;
		gActualMachineSpeed_FPM := gActualMachineSpeed_BPM*gRecipeActive.Repeat/12.0;

	(************************ AXIS VELOCITY MOVE **********************)

		MC_MoveVelocity_0.Axis:=gA[9].Ident;
		MC_MoveVelocity_0.Velocity:=gA[9].SP_Velocity*gA[9].AxisPeriod/60;
		MC_MoveVelocity_0.Acceleration:=gA[9].SP_Accel;
		MC_MoveVelocity_0.Deceleration:=gA[9].SP_Decel;
		MC_MoveVelocity_0.Direction:=mcPOSITIVE_DIR;
		IF ((EDGEPOS(gA[9].Cmd_ContinuousMotion)) OR (EDGEPOS(gA[9].Cmd_ContinuousMotionUpdate))) THEN
      MC_MoveVelocity_0.Execute:=1;
    ELSE
      MC_MoveVelocity_0.Execute := 0 ;
    END_IF;
		MC_MoveVelocity_0();

  (************************ AXIS HALT **********************)
    bAxisStop := NOT(gI_SafetyRelay_EStopOK)       OR
                 NOT(gGuardAlarmsOK)               OR
                 NOT(gBagMachine_WebBreakOK)       OR
                 gJog_Stop                         OR
                 NOT(gGeneralFaults_OK)            OR
                 NOT(gFastStop_OK)                 OR
                 ((gA[9].Ind_InMotion              OR
                   gA[9].Ind_ContinuousMotion)     AND
                  NOT(gA[9].Cmd_ContinuousMotion)  AND
                  NOT(gNormalStopReq))             ;

    MC_Halt_0.Axis:=gA[9].Ident;
    MC_Stop_0.Axis:=gA[9].Ident;
    IF bAxisStop                    AND
       ( gA[9].Ind_ContinuousMotion OR
         gA[9].Ind_DiscreteMotion ) THEN
        IF (NOT gI_SafetyRelay_EStopOK) THEN
          rDecelStop := gA[9].SP_EStopDecel ;
          MC_Stop_0.Deceleration := rDecelStop ;
          MC_Stop_0.Execute := 1 ;
          g_bIndStopFault := 1 ;
        ELSIF (NOT gGuardAlarmsOK) THEN
          rDecelStop:=gA[9].SP_GuardFaultDecel;
          g_bIndStopFault := 1 ;
        ELSIF (NOT gBagMachine_WebBreakOK) THEN
          rDecelStop:=gA[9].SP_WebBreakDecel;
          g_bIndStopFault := 1 ;
        ELSIF (NOT gGeneralFaults_OK) THEN
          rDecelStop:=gA[9].SP_GenFaultDecel;
          g_bIndStopFault := 1 ;
        ELSIF gJog_ToZeroSpeed THEN
          rDecelStop:=gA[9].SP_JogDecel;
        ELSIF (NOT gFastStop_OK) THEN
          rDecelStop:=gA[9].SP_FStopDecel;
        ELSE
          rDecelStop:=gA[9].SP_Decel;
        END_IF
      IF ( rDecelStop > rMemoDecelStop ) OR
         NOT(MC_Halt_0.Busy)             THEN
        IF MC_Halt_0.Busy THEN
          MC_Halt_0.Execute := 0 ;
          MC_Halt_0();
        END_IF
        MC_Halt_0.Execute := 1 ;
        MC_Halt_0.Deceleration := rDecelStop ;
        rMemoDecelStop := rDecelStop ;
      END_IF
    END_IF

    IF (MC_Halt_0.Done OR MC_Halt_0.CommandAborted OR MC_Halt_0.Error) THEN
      MC_Halt_0.Execute:=0;
      IF MC_Halt_0.Error THEN
        uiHalt_0_ErrorID := MC_Halt_0.ErrorID ;
        iHalt_0_ErrorCout := iHalt_0_ErrorCout + 1 ;
      END_IF
    END_IF

    IF (MC_Stop_0.Done OR MC_Stop_0.CommandAborted OR MC_Stop_0.Error) THEN
      MC_Stop_0.Execute:=0;
      IF MC_Stop_0.Error THEN
        uiStop_0_ErrorID := MC_Stop_0.ErrorID ;
        iStop_0_ErrorCout := iStop_0_ErrorCout + 1 ;
      END_IF
    END_IF
    MC_Stop_0();
    MC_Halt_0();

    IF NOT(MC_Stop_0.Busy) AND
       NOT(MC_Halt_0.Busy) AND
       1                   THEN
      g_bIndStopFault := 0 ;
    END_IF

	//************************ AXIS STOP ON POSITION **********************
  bAxisStopPos := NOT(MC_Halt_0.Busy)        AND
                  NOT(MC_Stop_0.Busy)        AND
                  gA[9].Ind_ContinuousMotion AND
                  gNormalStopReq             ;

    // Stop position calculation
    // Stop position = Perf in park position and tearing not in contact zone
    IF bAxisStopPos THEN
      IF NOT(MC_MoveAbsolute_0.Execute)THEN
        // Position on Master in Deg when Perf is in park position
        rTempCalc_[0] := g_rPosParkMasterCam - gRecipeActive.Perf_Offset/gRecipeActive.Repeat * 360.0 ;
        rPosMaPerfPark := H_FC_Modulus (
                               IN_rMod := 360,
                               IN_rVar := rTempCalc_[0]
                                       ) ;

        // Zone Master when Tearing Axis is in contact zone
        // Pos beginning ( Pos of the beginning of the contact zone on tearing axis = 0° )
        rPosMaTearInContactZ_Beg := 360 - gA[4].rActPhasDeg ;
        // Pos end  ( Pos of the end of the contact zone on tearing axis = gr_rTearAxContactZone° )
        rPosMaTearInContactZ_End := gr_rTearAxContactZone + rPosMaTearInContactZ_Beg ;

        // Correction if master stop whith Tearing in contact zone in case of RS15
        IF g_iMachType = C_iRS15 THEN
          IF ( rPosMaTearInContactZ_Beg < rPosMaTearInContactZ_End ) THEN
            IF ( rPosMaPerfPark > rPosMaTearInContactZ_Beg ) AND
               ( rPosMaPerfPark < rPosMaTearInContactZ_End ) THEN
              rPosMaPerfPark := rPosMaTearInContactZ_End ;
            END_IF
          ELSE
            IF ( rPosMaPerfPark > rPosMaTearInContactZ_Beg ) OR
               ( rPosMaPerfPark < rPosMaTearInContactZ_End ) THEN
              rPosMaPerfPark := rPosMaTearInContactZ_End ;
            END_IF
          END_IF
        END_IF
      END_IF
      gStopPosition := H_FC_Modulus (
                            IN_rMod := 360,
                            IN_rVar := rPosMaPerfPark
                                    ) ;
			MC_MoveAbsolute_0.Velocity := gActualMachineSpeed_BPM * gA[9].AxisPeriod/60;
			MC_MoveAbsolute_0.Execute:=1;
		END_IF
		MC_MoveAbsolute_0.Deceleration:=gA[9].SP_Decel;
		MC_MoveAbsolute_0.Acceleration:=gA[9].SP_Accel;
		MC_MoveAbsolute_0.Direction := mcPOSITIVE_DIR;
		MC_MoveAbsolute_0.Axis := gA[9].Ident;
		MC_MoveAbsolute_0.Position := gStopPosition*gA[9].UnitsPerDeg;
		IF (MC_MoveAbsolute_0.Done OR MC_MoveAbsolute_0.CommandAborted OR MC_MoveAbsolute_0.Error) THEN
			ErrorID := MC_MoveAbsolute_0.ErrorID;
			MC_MoveAbsolute_0.Execute:=0;
		END_IF
    MC_MoveAbsolute_0();
	END_IF

END_PROGRAM
```

#### A9_Basic.var - Local variables
```iecst
(********************************************************************
 * COPYRIGHT -- Microsoft
 ********************************************************************
 * Program: A9_Basic
 * File: A9_Basic.var
 * Author: pkiel
 * Created: July 12, 2011
 ********************************************************************
 * Local variables of program A9_Basic
 ********************************************************************)
VAR
	AutoAck : BOOL;
	AxisErrorNcAccess : UINT;
	DriveStatus : MC_DRIVESTATUS_TYP;
	ErrorID : UINT;
	HomeRestore : BOOL;
	InitEndlessPosition : BOOL;
	InitModPos_Done : BOOL;
	InitModPosition : BOOL;
	MC_BR_InitEndlessPosition_0 : MC_BR_InitEndlessPosition;
	MC_BR_InitModPos_0 : MC_BR_InitModPos;
	MC_BR_ReadDriveStatus_0 : MC_BR_ReadDriveStatus;
	MC_Home_0 : MC_Home;
	MC_Home_1 : MC_Home;
	MC_MoveAbsolute_0 : MC_MoveAbsolute;
	MC_MoveVelocity_0 : MC_MoveVelocity;
	MC_ReadActualPosition_0 : MC_ReadActualPosition;
	MC_ReadActualVelocity_0 : MC_ReadActualVelocity;
	MC_ReadAxisError_0 : MC_ReadAxisError;
	MC_ReadStatus_0 : MC_ReadStatus;
	MC_Reset_0 : MC_Reset;
  MC_Stop_0 : MC_Stop;
  uiStop_0_ErrorID : UINT ;
  iStop_0_ErrorCout : INT ;
  MC_Halt_0 : MC_Halt;
  uiHalt_0_ErrorID : UINT ;
  iHalt_0_ErrorCout : INT ;
  rDecelStop     : REAL ;
  rMemoDecelStop : REAL ;
	ResetError : BOOL;
  rPosMaPerfPark : REAL ; (*Pos on Master Perf in park position, in Deg*)
  rPosMaTearInContactZ_Beg : REAL ; (*Pos on Master beginning of the tearing contact zone, in Deg*)
  rPosMaTearInContactZ_End : REAL ; (*Pos on Master end of the tearing contact zone, in Deg*)
  rTravelMaEndContactZ : REAL ;
  rTempCalc_ : ARRAY[0..9] OF REAL ;
  bAxisStop : BOOL ;
  bAxisStopPos : BOOL ;
  bTest_ : ARRAY[0..9] OF BOOL;
  iTest_ : ARRAY[0..9] OF INT;
  iTestTrac : INT ;
  stTON_0 : TON ;
  stTON_1 : TON ;

END_VAR
```

### Program Logical/BagMachine_Section/MasterAxis/A9_Init/A9_Control (IEC) - Servo Control

#### A9_ControlCyclic.ld - Cyclic code
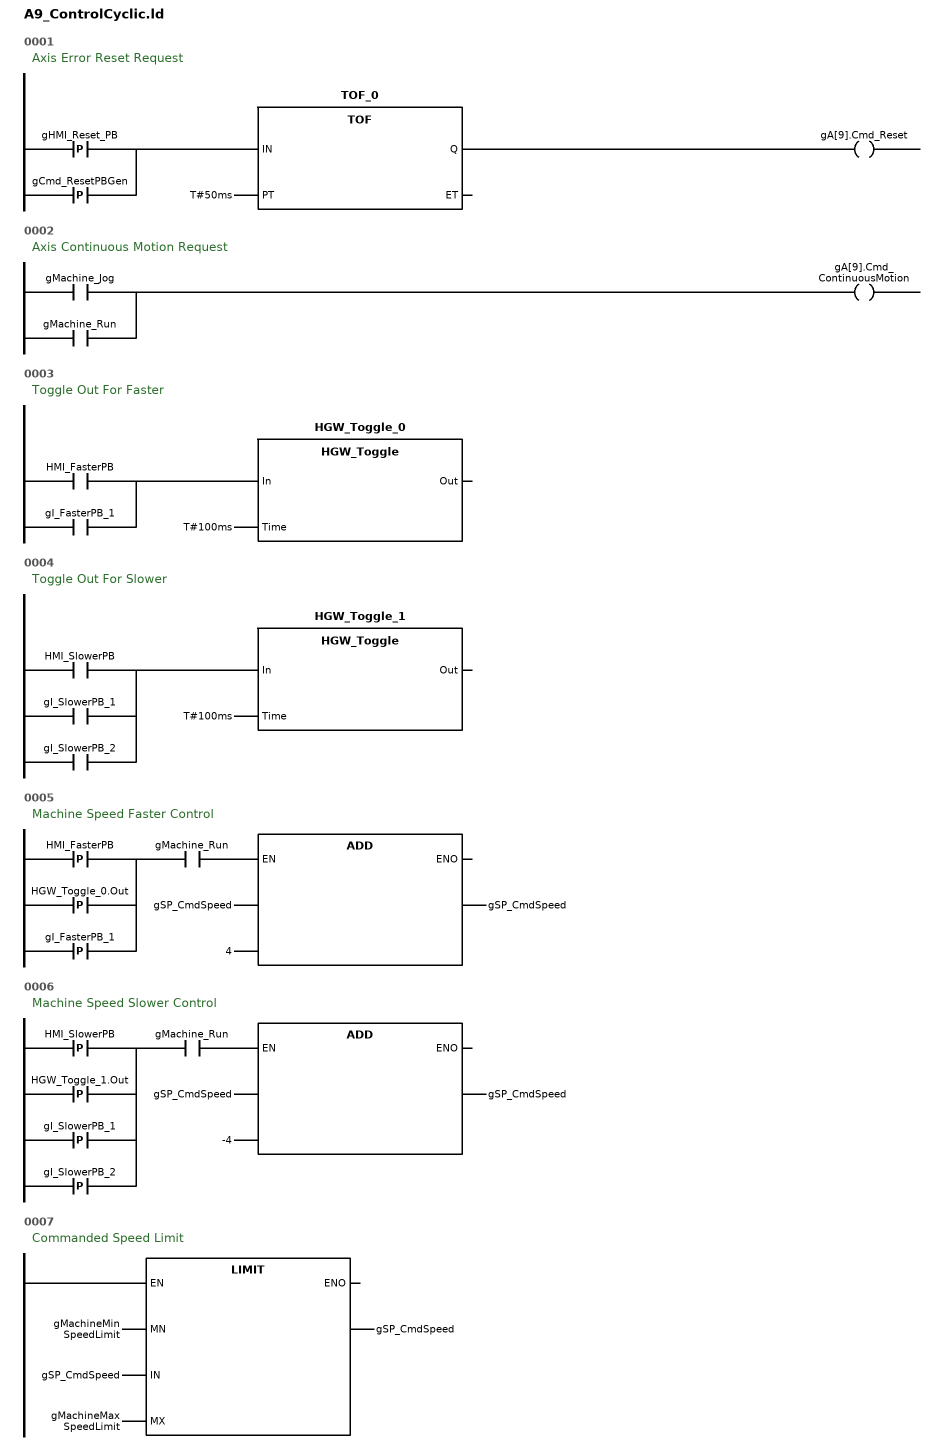
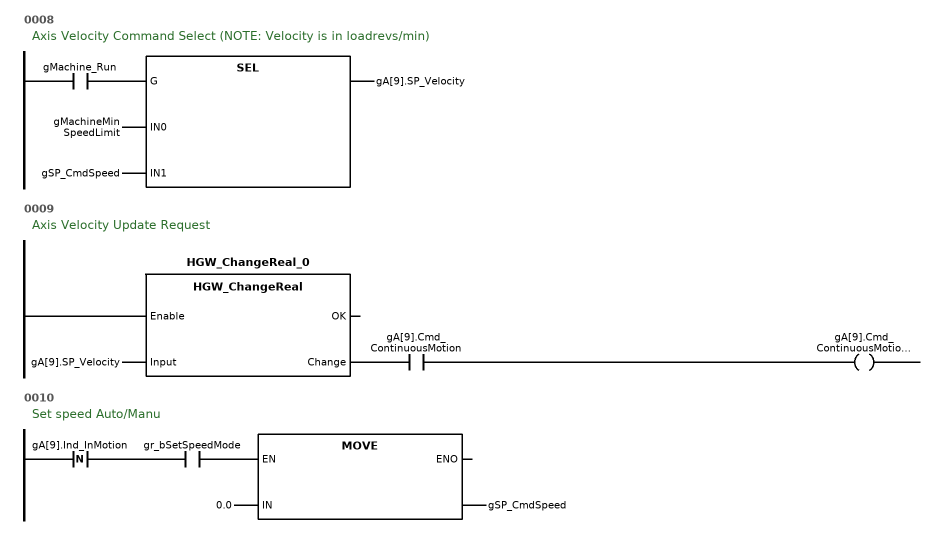
Ladder, written as Structured Text:
```iecst
(********************************************************************
 * COPYRIGHT -- Microsoft
 ********************************************************************
 * Program: A9_Control
 * File: A9_ControlCyclic.ld
 * Author: pkiel
 * Created: July 12, 2011
 ********************************************************************
 * Implementation of program A9_Control
 ********************************************************************)

PROGRAM _CYCLIC
VAR
    _e1 : R_TRIG;
    _e2 : R_TRIG;
    _e3 : R_TRIG;
    _e4 : R_TRIG;
    _e5 : R_TRIG;
    _e6 : R_TRIG;
    _e7 : R_TRIG;
    _e8 : R_TRIG;
    _e9 : R_TRIG;
    _e10 : F_TRIG;
END_VAR
(* Network 1: Axis Error Reset Request *)
_e1(CLK := gHMI_Reset_PB);
_e2(CLK := gCmd_ResetPBGen);
TOF_0(IN := _e1.Q OR _e2.Q, PT := T#50ms);
gA[9].Cmd_Reset := TOF_0.Q;

(* Network 2: Axis Continuous Motion Request *)
gA[9].Cmd_ContinuousMotion := gMachine_Jog OR gMachine_Run;

(* Network 3: Toggle Out For Faster *)
HGW_Toggle_0(In := HMI_FasterPB OR gI_FasterPB_1, Time := T#100ms);

(* Network 4: Toggle Out For Slower *)
HGW_Toggle_1(In := HMI_SlowerPB OR gI_SlowerPB_1 OR gI_SlowerPB_2, Time := T#100ms);

(* Network 5: Machine Speed Faster Control *)
_e3(CLK := HMI_FasterPB);
_e4(CLK := HGW_Toggle_0.Out);
_e5(CLK := gI_FasterPB_1);
IF (_e3.Q OR _e4.Q OR _e5.Q) AND gMachine_Run THEN gSP_CmdSpeed := gSP_CmdSpeed + 4; END_IF;

(* Network 6: Machine Speed Slower Control *)
_e6(CLK := HMI_SlowerPB);
_e7(CLK := HGW_Toggle_1.Out);
_e8(CLK := gI_SlowerPB_1);
_e9(CLK := gI_SlowerPB_2);
IF (_e6.Q OR _e7.Q OR _e8.Q OR _e9.Q) AND gMachine_Run THEN gSP_CmdSpeed := gSP_CmdSpeed + -4; END_IF;

(* Network 7: Commanded Speed Limit *)
gSP_CmdSpeed := LIMIT(MN := gMachineMinSpeedLimit, IN := gSP_CmdSpeed, MX := gMachineMaxSpeedLimit);

(* Network 8: Axis Velocity Command Select (NOTE: Velocity is in loadrevs/min) *)
gA[9].SP_Velocity := SEL(G := gMachine_Run, IN0 := gMachineMinSpeedLimit, IN1 := gSP_CmdSpeed);

(* Network 9: Axis Velocity Update Request *)
HGW_ChangeReal_0(Enable := TRUE, Input := gA[9].SP_Velocity);
gA[9].Cmd_ContinuousMotionUpdate := HGW_ChangeReal_0.Change AND gA[9].Cmd_ContinuousMotion;

(* Network 10: Set speed Auto/Manu *)
_e10(CLK := gA[9].Ind_InMotion);
IF _e10.Q AND gr_bSetSpeedMode THEN gSP_CmdSpeed := 0.0; END_IF;
END_PROGRAM
```

#### A9_Control.var - Local variables
```iecst
(********************************************************************
 * COPYRIGHT -- Microsoft
 ********************************************************************
 * Program: A9_Control
 * File: A9_Control.var
 * Author: pkiel
 * Created: July 12, 2011
 ********************************************************************
 * Local variables of program A9_Control
 ********************************************************************)
VAR
	HGW_ChangeReal_0 : HGW_ChangeReal;
	HGW_Toggle_0 : HGW_Toggle;
	HGW_Toggle_1 : HGW_Toggle;
	HMI_FasterPB : BOOL;
  HMI_SlowerPB : BOOL;
  HMI_b : BOOL;
	TOF_0 : TOF;
END_VAR

VAR RETAIN
END_VAR
```

### Program Logical/BagMachine_Section/MasterAxis/A9_Init/SetSpeedMode (IEC) - A new program

#### SetSpeedMode.var - Local variables
```iecst
(********************************************************************
 * COPYRIGHT -- .
 ********************************************************************
 * Program: SetSpeedMode
 * File: SetSpeedMode.var
 * Author: dominique
 * Created: September 29, 2011
 ********************************************************************
 * Local variables of program SetSpeedMode
 ********************************************************************)

VAR
  HMI_uiConfirmSetSpeedVisibl : UINT ;
  HMI_bSetSpeed_PB : BOOL ;
END_VAR

VAR RETAIN
END_VAR
```

- Data object Logical/BagMachine_Section/Perf/CamProfTest (Cam) - ACP10: Cam Profile data object. (no source held here)

### Program Logical/BagMachine_Section/Perf/Perf_Gen (IEC) - General Perf Control

#### Perf_GenCyclic.st - Cyclic code
```iecst
(********************************************************************
 * COPYRIGHT -- Microsoft
 ********************************************************************
 * Program: Perf_Gen
 * File: Perf_GenCyclic.st
 * Author: pkiel
 * Created: July 19, 2011
 ********************************************************************
 * Implementation of program Perf_Gen
 ********************************************************************)

PROGRAM _CYCLIC

(* Perf Off/On From HMI *)
	HGW_2StatePB_0.PB := EDGEPOS(Perf_PB AND NOT gA[9].Ind_InMotion);
	PerfText_Ind := HGW_2StatePB_0.Text_Ind;
	PerfColor_Ind := HGW_2StatePB_0.Color_Ind;
	gPerf_On := HGW_2StatePB_0.State1;
	HGW_2StatePB_0();

  IF gPerf_ParkRequired THEN
    H_FB_Flash_0(IN_bEnable:=1, IN_rNumFlashPerSec:=1.0) ;
    IF H_FB_Flash_0.OUT_bFlash THEN
      PerfColor_Ind := gBlue + gWhite * 256 ;
    ELSE
      PerfColor_Ind := gGreen + gBlack * 256 ;
    END_IF
  ELSE
    H_FB_Flash_0(IN_bEnable:=0, IN_rNumFlashPerSec:=1.0) ;
  END_IF

(* Is Perf Park Required *)
	IF (EDGENEG(gPerf_On) AND NOT InParkPosition) THEN
		gPerf_ParkRequired :=1;
	END_IF
	IF (EDGEPOS(gPerf_On)) THEN
		gPerf_ParkRequired :=0;
	END_IF

(* Perf In Park Position *)
  rTempPosA1_Deg := H_FC_Modulus(IN_rMod:=360/gSP_PerfKnifeCount, IN_rVar:=gA[1].PositionDeg) ;
	IF (rTempPosA1_Deg>(gSP_A[1].ParkPosition-2.0)) AND (rTempPosA1_Deg<(gSP_A[1].ParkPosition+2.0)) THEN
		InParkPosition := 1;
	ELSE
		InParkPosition := 0;
	END_IF
	TON_0(IN := InParkPosition, PT := T#2s);
	IF(InParkPosition AND TON_0.Q AND NOT gPerf_On) THEN
		gPerf_ParkRequired := 0;
  END_IF

  // Limit IHM Perf Set Up values
  // Envelope Bag Perf
  g_rSizeEnvBPerf_mm        := LIMIT(g_rMaxBagSize_EnvB_mm/25.4,gRecipeActive.rEnvB_PerfSize_in,g_rMinBagSize_EnvB_mm/25.4) ;
  gSP_EnvBPerf.HomeOffset   := LIMIT(0.0,gSP_EnvBPerf.HomeOffset,360.0) ;
  gSP_EnvBPerf.MatchedSpeed := LIMIT(0.0,gSP_EnvBPerf.MatchedSpeed,360.0) ;
  gSP_EnvBPerf.ParkPosition := LIMIT(0.0,gSP_EnvBPerf.ParkPosition,360.0) ;
  // Standard Perf
  gSP_StandPerf.HomeOffset   := LIMIT(0.0,gSP_StandPerf.HomeOffset,360.0) ;
  gSP_StandPerf.MatchedSpeed := LIMIT(0.0,gSP_StandPerf.MatchedSpeed,360.0) ;
  gSP_StandPerf.ParkPosition := LIMIT(0.0,gSP_StandPerf.ParkPosition,360.0) ;

(* Theoretical Perimeter...Large Cylinder = 400mm (15.748") , Small Cylinder = 270mm (10.630") *)
	RepeatMetric := REAL_TO_INT(gRecipeActive.Repeat*25.4);
  IF g_rSizeSPerf_mm > 0.0 AND
     g_rSizeLPerf_mm > 0.0 THEN

    IF NOT(gRecipeActive.bSelEnvBProd) THEN
    	IF (gSP_PerfCylSelect=0) THEN  (* Small Cylinder *)
        g_rActualSizePerf_in := g_rSizeSPerf_mm/25.4 ;
        g_iPerfType := 0 ;
    		IF (RepeatMetric<=g_rBagSize1to2SPerf_mm) THEN
    			gSP_PerfKnifeCount     := 2;
    			SecondKnife_Visibility := 0;
    		ELSE
    			gSP_PerfKnifeCount     := 1;
    			SecondKnife_Visibility := 1;
    		END_IF
    	ELSE  (* Large Cylinder *)
        g_rActualSizePerf_in := g_rSizeLPerf_mm/25.4 ;
        g_iPerfType := 1 ;
    		IF (RepeatMetric<=g_rBagSize1to2LPerf_mm) THEN
    			gSP_PerfKnifeCount := 2;
    			SecondKnife_Visibility := 0;
    		ELSE
    			gSP_PerfKnifeCount     := 1;
    			SecondKnife_Visibility := 1;
    		END_IF
      END_IF

      // Perf Set Up
      gSP_StandPerf.HomeOffset   := 90.0 + gSP_StandPerf.rZoneBefPerf_in/g_rActualSizePerf_in * 360.0 ; // D.M. Le 10/01/2012 Pyrollpack_14661   Because operator is able to change the size of the Perf => Easier for operator to set automatically these values
      gSP_StandPerf.ParkPosition := gSP_StandPerf.HomeOffset ;
      gSP_A[1].HomeOffset        := gSP_StandPerf.HomeOffset ;
      gSP_A[1].ParkPosition      := gSP_StandPerf.ParkPosition ;
      gSP_A[1].MatchedSpeed      := (gSP_StandPerf.rZoneBefPerf_in+gSP_StandPerf.rZoneAftPerf_in)/g_rActualSizePerf_in * 360.0 ;
    ELSE   // Case Envelope Bag
      g_rActualSizePerf_in := gRecipeActive.rEnvB_PerfSize_in ;
      gSP_PerfKnifeCount     := 1;  // Always 1 knife only
      SecondKnife_Visibility := 1;
      g_iPerfType := 2 ;

      // Perf Set Up
      gSP_EnvBPerf.HomeOffset   := 90.0 + gSP_EnvBPerf.rZoneBefPerf_in/g_rActualSizePerf_in * 360.0 ; // D.M. Le 10/01/2012 Pyrollpack_14661   Because operator is able to change the size of the Perf => Easier for operator to set automatically these values
      gSP_EnvBPerf.ParkPosition := gSP_EnvBPerf.HomeOffset ;
      gSP_A[1].HomeOffset       := gSP_EnvBPerf.HomeOffset ;
      gSP_A[1].ParkPosition     := gSP_EnvBPerf.ParkPosition ;
      gSP_A[1].MatchedSpeed     := (gSP_EnvBPerf.rZoneBefPerf_in+gSP_EnvBPerf.rZoneAftPerf_in)/g_rActualSizePerf_in * 360.0 ;
    END_IF
  END_IF

  gA[1].UnitsPerInch := gA[1].AxisPeriod/g_rActualSizePerf_in ;
  gA[1].InchPerDeg   := g_rActualSizePerf_in / 360 ;

  // Perf Set Up visibility
  IF (g_iPerfType <= 1) THEN
    HMI_iEnvBPerfSetUpVisible := 1 ;  // Envelope Bag unvisible
    HMI_iPerfSetUpVisible     := 0 ;  // Standard Bag visible
  ELSE
    HMI_iEnvBPerfSetUpVisible := 0 ;  // Envelope Bag visible
    HMI_iPerfSetUpVisible     := 1 ;  // Standard Bag unvisible
  END_IF

END_PROGRAM
```

#### Perf_GenInit.st - Initialization code
```iecst
(********************************************************************
 * COPYRIGHT -- Microsoft
 ********************************************************************
 * Program: Perf_Gen
 * File: Perf_GenInit.st
 * Author: pkiel
 * Created: July 19, 2011
 ********************************************************************
 * Implementation of program Perf_Gen
 ********************************************************************)

PROGRAM _INIT

(* Perf Off/On PB Colors *)
	HGW_2StatePB_0.BackColor_State0 := gBlue;
	HGW_2StatePB_0.ForeColor_State0 := gWhite;
	HGW_2StatePB_0.BackColor_State1 := gGreen;
	HGW_2StatePB_0.ForeColor_State1 := gBlack;

END_PROGRAM
```

- Data object Logical/BagMachine_Section/Perf/Axis1/A1_Init (Ax) - Servo Axis Initialization File (no source held here)

### Program Logical/BagMachine_Section/Perf/Axis1/A1_Basic (IEC) - Basic Servo

#### A1_BasicInit.st
```iecst
(********************************************************************
 * COPYRIGHT -- Microsoft
 ********************************************************************
 * Program: A1_Basic
 * File: A1_BasicInit.st
 * Author: pkiel
 * Created: July 11, 2011
 ********************************************************************
 * Implementation of program A1_Basic
 ********************************************************************)

PROGRAM _INIT

	(* Axis Setpoint Variables *)
		gA[1].SP_MotorPPR := 18000;
		gA[1].SP_GearBoxInput:= 2;
		gA[1].SP_GearBoxOutput:= 1;
		gA[1].AxisPeriod := (gA[1].SP_MotorPPR*gA[1].SP_GearBoxInput/gA[1].SP_GearBoxOutput);
		gA[1].UnitsPerDeg := gA[1].AxisPeriod/360;
		gA[1].SP_Accel := 0.2*gA[1].AxisPeriod;
		gA[1].SP_Decel := 0.4*gA[1].AxisPeriod;
		gA[1].SP_EStopDecel := 1000.0*gA[1].AxisPeriod; // Stop axis from 1000 tr/min in 1s
    gA[1].rSP_CorPosVel := 0.0 ;
    gA[1].rSP_CorPosVel := 0.0 ;
    gA[1].rSP_OverrideV := 1.0 ;
    gA[1].rSP_OverrideA := 1.0 ;
    gA[1].Cmd_EStopDisable := 0 ;

	(* access master axis *)
		AxisErrorNcAccess := ncaccess(ncACP10MAN, ADR('Axis1'), ADR(gA[1].Ident));

	(* Trigger Initialization Of ModPosition *)
		InitModPosition:=1;

END_PROGRAM
```

### Program Logical/BagMachine_Section/Perf/Axis1/A1_Control (IEC) - Servo Control
